// Functions/Basic Container Operations/F_VN_GetAt/F_VN_GetAt_TcVnVector4_UINT

	{attribute 'TcIecLibraryType'}
	{attribute 'external_name' := 'F_VN_GetAt_TcVnVector4_UINT_GUID_DACA282F_CF71_0B71_5078_D95B06B34C79'}
	(* Gets the TcVnVector4_UINT element at the specified index of the container. *)
	FUNCTION F_VN_GetAt_TcVnVector4_UINT : HRESULT
	VAR_INPUT
		ipContainer	:	ITcVnContainer;	(* Container with TcVnVector4_UINT elements *)
		aElement	:	REFERENCE TO TcVnVector4_UINT;	(* Returns the element at the specified index *)
		nIndex	:	ULINT;	(* Index of the requested element *)
		hrPrev	:	HRESULT;	(* HRESULT indicating the result of previous operations (If SUCCEEDED(hrPrev) equals false, no operation is executed.) *)
	END_VAR

END_FUNCTION

// Functions/Basic Container Operations/F_VN_GetAt/F_VN_GetAt_TcVnVector4_USINT

	{attribute 'TcIecLibraryType'}
	{attribute 'external_name' := 'F_VN_GetAt_TcVnVector4_USINT_GUID_B04CDEB5_6B6C_0BE2_4BEB_6EA1CC43E558'}
	(* Gets the TcVnVector4_USINT element at the specified index of the container. *)
	FUNCTION F_VN_GetAt_TcVnVector4_USINT : HRESULT
	VAR_INPUT
		ipContainer	:	ITcVnContainer;	(* Container with TcVnVector4_USINT elements *)
		aElement	:	REFERENCE TO TcVnVector4_USINT;	(* Returns the element at the specified index *)
		nIndex	:	ULINT;	(* Index of the requested element *)
		hrPrev	:	HRESULT;	(* HRESULT indicating the result of previous operations (If SUCCEEDED(hrPrev) equals false, no operation is executed.) *)
	END_VAR

END_FUNCTION

// Functions/Basic Container Operations/F_VN_GetAt/F_VN_GetAt_UDINT

	{attribute 'TcIecLibraryType'}
	{attribute 'external_name' := 'F_VN_GetAt_UDINT_GUID_BF979232_2744_07C5_6489_84B0C61F3275'}
	(* Gets the UDINT element at the specified index of the container. *)
	FUNCTION F_VN_GetAt_UDINT : HRESULT
	VAR_INPUT
		ipContainer	:	ITcVnContainer;	(* Container with UDINT elements *)
		nElement	:	REFERENCE TO UDINT;	(* Returns the element at the specified index *)
		nIndex	:	ULINT;	(* Index of the requested element *)
		hrPrev	:	HRESULT;	(* HRESULT indicating the result of previous operations (If SUCCEEDED(hrPrev) equals false, no operation is executed.) *)
	END_VAR

END_FUNCTION

// Functions/Basic Container Operations/F_VN_GetAt/F_VN_GetAt_UINT

	{attribute 'TcIecLibraryType'}
	{attribute 'external_name' := 'F_VN_GetAt_UINT_GUID_D4F7DF25_3651_0BE4_4285_2E117680DE7D'}
	(* Gets the UINT element at the specified index of the container. *)
	FUNCTION F_VN_GetAt_UINT : HRESULT
	VAR_INPUT
		ipContainer	:	ITcVnContainer;	(* Container with UINT elements *)
		nElement	:	REFERENCE TO UINT;	(* Returns the element at the specified index *)
		nIndex	:	ULINT;	(* Index of the requested element *)
		hrPrev	:	HRESULT;	(* HRESULT indicating the result of previous operations (If SUCCEEDED(hrPrev) equals false, no operation is executed.) *)
	END_VAR

END_FUNCTION

// Functions/Basic Container Operations/F_VN_GetAt/F_VN_GetAt_ULINT

	{attribute 'TcIecLibraryType'}
	{attribute 'external_name' := 'F_VN_GetAt_ULINT_GUID_BCB044E1_AE9F_0A92_654C_54D02EC2BF64'}
	(* Gets the ULINT element at the specified index of the container. *)
	FUNCTION F_VN_GetAt_ULINT : HRESULT
	VAR_INPUT
		ipContainer	:	ITcVnContainer;	(* Container with ULINT elements *)
		nElement	:	REFERENCE TO ULINT;	(* Returns the element at the specified index *)
		nIndex	:	ULINT;	(* Index of the requested element *)
		hrPrev	:	HRESULT;	(* HRESULT indicating the result of previous operations (If SUCCEEDED(hrPrev) equals false, no operation is executed.) *)
	END_VAR

END_FUNCTION

// Functions/Basic Container Operations/F_VN_GetAt/F_VN_GetAt_USINT

	{attribute 'TcIecLibraryType'}
	{attribute 'external_name' := 'F_VN_GetAt_USINT_GUID_3E49D359_324C_0975_751E_A652C8C9EF75'}
	(* Gets the USINT element at the specified index of the container. *)
	FUNCTION F_VN_GetAt_USINT : HRESULT
	VAR_INPUT
		ipContainer	:	ITcVnContainer;	(* Container with USINT elements *)
		nElement	:	REFERENCE TO USINT;	(* Returns the element at the specified index *)
		nIndex	:	ULINT;	(* Index of the requested element *)
		hrPrev	:	HRESULT;	(* HRESULT indicating the result of previous operations (If SUCCEEDED(hrPrev) equals false, no operation is executed.) *)
	END_VAR

END_FUNCTION

// Functions/Basic Container Operations/F_VN_InsertIntoContainer/F_VN_InsertIntoContainer_ITcVnContainer

	{attribute 'TcIecLibraryType'}
	{attribute 'external_name' := 'F_VN_InsertIntoContainer_ITcVnContainer_GUID_A60BDE14_E4D7_0797_570B_140C623D0487'}
	(* Insert an element (or a range of elements) into a container before the specified position. *)
	FUNCTION F_VN_InsertIntoContainer_ITcVnContainer : HRESULT
	VAR_INPUT
		ipElement	:	ITcVnContainer;	(* Single element to insert into ipContainer or container with several elements *)
		ipContainer	:	ITcVnContainer;	(* Container in which to insert the element *)
		nIndex	:	ULINT;	(* Position, before which the element will be inserted *)
		hrPrev	:	HRESULT;	(* HRESULT indicating the result of previous operations (If SUCCEEDED(hrPrev) equals false, no operation is executed.) *)
	END_VAR

END_FUNCTION

// Functions/Basic Container Operations/F_VN_InsertIntoContainer/F_VN_InsertIntoContainer_ITcVnForwardIterator

	{attribute 'TcIecLibraryType'}
	{attribute 'external_name' := 'F_VN_InsertIntoContainer_ITcVnForwardIterator_GUID_FB7539B3_B7C2_0135_5324_E11529024484'}
	(* Insert an element (represented by an iterator) into a container before the specified position. *)
	FUNCTION F_VN_InsertIntoContainer_ITcVnForwardIterator : HRESULT
	VAR_INPUT
		ipElement	:	ITcVnForwardIterator;	(* Single element to insert into ipContainer *)
		ipContainer	:	ITcVnContainer;	(* Container in which to insert the element *)
		nIndex	:	ULINT;	(* Position, before which the element will be inserted *)
		hrPrev	:	HRESULT;	(* HRESULT indicating the result of previous operations (If SUCCEEDED(hrPrev) equals false, no operation is executed.) *)
	END_VAR

END_FUNCTION

// Functions/Basic Container Operations/F_VN_InsertIntoContainer/F_VN_InsertIntoContainer_DINT

	{attribute 'TcIecLibraryType'}
	{attribute 'external_name' := 'F_VN_InsertIntoContainer_DINT_GUID_9477BFDC_23EB_04A7_4507_F78D3CC46D82'}
	(* Insert an element of type DINT into a container before the specified position. *)
	FUNCTION F_VN_InsertIntoContainer_DINT : HRESULT
	VAR_INPUT
		nElement	:	DINT;	(* Single element to insert into ipContainer *)
		ipContainer	:	ITcVnContainer;	(* Container in which to insert the element *)
		nIndex	:	ULINT;	(* Position, before which the element will be inserted *)
		hrPrev	:	HRESULT;	(* HRESULT indicating the result of previous operations (If SUCCEEDED(hrPrev) equals false, no operation is executed.) *)
	END_VAR

END_FUNCTION

// Functions/Basic Container Operations/F_VN_InsertIntoContainer/F_VN_InsertIntoContainer_INT

	{attribute 'TcIecLibraryType'}
	{attribute 'external_name' := 'F_VN_InsertIntoContainer_INT_GUID_6C53FE75_6CDB_00E0_52DC_8EED063716A2'}
	(* Insert an element of type INT into a container before the specified position. *)
	FUNCTION F_VN_InsertIntoContainer_INT : HRESULT
	VAR_INPUT
		nElement	:	INT;	(* Single element to insert into ipContainer *)
		ipContainer	:	ITcVnContainer;	(* Container in which to insert the element *)
		nIndex	:	ULINT;	(* Position, before which the element will be inserted *)
		hrPrev	:	HRESULT;	(* HRESULT indicating the result of previous operations (If SUCCEEDED(hrPrev) equals false, no operation is executed.) *)
	END_VAR

END_FUNCTION

// Functions/Basic Container Operations/F_VN_InsertIntoContainer/F_VN_InsertIntoContainer_ITcVnImage

	{attribute 'TcIecLibraryType'}
	{attribute 'external_name' := 'F_VN_InsertIntoContainer_ITcVnImage_GUID_818AAE11_662C_0FFE_6EFF_8404FD801653'}
	(* Insert an element of type ITcVnImage into a container before the specified position. *)
	FUNCTION F_VN_InsertIntoContainer_ITcVnImage : HRESULT
	VAR_INPUT
		ipElement	:	ITcVnImage;	(* Single element to insert into ipContainer *)
		ipContainer	:	ITcVnContainer;	(* Container in which to insert the element *)
		nIndex	:	ULINT;	(* Position, before which the element will be inserted *)
		hrPrev	:	HRESULT;	(* HRESULT indicating the result of previous operations (If SUCCEEDED(hrPrev) equals false, no operation is executed.) *)
	END_VAR

END_FUNCTION

// Functions/Basic Container Operations/F_VN_InsertIntoContainer/F_VN_InsertIntoContainer_LREAL

	{attribute 'TcIecLibraryType'}
	{attribute 'external_name' := 'F_VN_InsertIntoContainer_LREAL_GUID_096F557A_3F3F_05E3_5F27_949C48CD0B7C'}
	(* Insert an element of type LREAL into a container before the specified position. *)
	FUNCTION F_VN_InsertIntoContainer_LREAL : HRESULT
	VAR_INPUT
		fElement	:	LREAL;	(* Single element to insert into ipContainer *)
		ipContainer	:	ITcVnContainer;	(* Container in which to insert the element *)
		nIndex	:	ULINT;	(* Position, before which the element will be inserted *)
		hrPrev	:	HRESULT;	(* HRESULT indicating the result of previous operations (If SUCCEEDED(hrPrev) equals false, no operation is executed.) *)
	END_VAR

END_FUNCTION

// Functions/Basic Container Operations/F_VN_InsertIntoContainer/F_VN_InsertIntoContainer_REAL

	{attribute 'TcIecLibraryType'}
	{attribute 'external_name' := 'F_VN_InsertIntoContainer_REAL_GUID_45718397_CD8F_043C_4B3C_FAEFC2A76FAA'}
	(* Insert an element of type REAL into a container before the specified position. *)
	FUNCTION F_VN_InsertIntoContainer_REAL : HRESULT
	VAR_INPUT
		fElement	:	REAL;	(* Single element to insert into ipContainer *)
		ipContainer	:	ITcVnContainer;	(* Container in which to insert the element *)
		nIndex	:	ULINT;	(* Position, before which the element will be inserted *)
		hrPrev	:	HRESULT;	(* HRESULT indicating the result of previous operations (If SUCCEEDED(hrPrev) equals false, no operation is executed.) *)
	END_VAR

END_FUNCTION

// Functions/Basic Container Operations/F_VN_InsertIntoContainer/F_VN_InsertIntoContainer_SINT

	{attribute 'TcIecLibraryType'}
	{attribute 'external_name' := 'F_VN_InsertIntoContainer_SINT_GUID_A7FF57E5_5EEA_0357_45DF_3CF7D68E66D8'}
	(* Insert an element of type SINT into a container before the specified position. *)
	FUNCTION F_VN_InsertIntoContainer_SINT : HRESULT
	VAR_INPUT
		nElement	:	SINT;	(* Single element to insert into ipContainer *)
		ipContainer	:	ITcVnContainer;	(* Container in which to insert the element *)
		nIndex	:	ULINT;	(* Position, before which the element will be inserted *)
		hrPrev	:	HRESULT;	(* HRESULT indicating the result of previous operations (If SUCCEEDED(hrPrev) equals false, no operation is executed.) *)
	END_VAR

END_FUNCTION

// Functions/Basic Container Operations/F_VN_InsertIntoContainer/F_VN_InsertIntoContainer_TcVnDMatch

	{attribute 'TcIecLibraryType'}
	{attribute 'external_name' := 'F_VN_InsertIntoContainer_TcVnDMatch_GUID_195FA26A_4C98_0C0C_6341_BCA50298A1E2'}
	(* Insert an element of type TcVnDMatch into a container before the specified position. *)
	FUNCTION F_VN_InsertIntoContainer_TcVnDMatch : HRESULT
	VAR_INPUT
		stElement	:	REFERENCE TO TcVnDMatch;	(* Single element to insert into ipContainer *)
		ipContainer	:	ITcVnContainer;	(* Container in which to insert the element *)
		nIndex	:	ULINT;	(* Position, before which the element will be inserted *)
		hrPrev	:	HRESULT;	(* HRESULT indicating the result of previous operations (If SUCCEEDED(hrPrev) equals false, no operation is executed.) *)
	END_VAR

END_FUNCTION

// Functions/Basic Container Operations/F_VN_InsertIntoContainer/F_VN_InsertIntoContainer_TcVnKeyPoint

	{attribute 'TcIecLibraryType'}
	{attribute 'external_name' := 'F_VN_InsertIntoContainer_TcVnKeyPoint_GUID_CDF375E9_8EF3_01A8_6EAB_4A74123B3E8C'}
	(* Insert an element of type TcVnKeyPoint into a container before the specified position. *)
	FUNCTION F_VN_InsertIntoContainer_TcVnKeyPoint : HRESULT
	VAR_INPUT
		stElement	:	REFERENCE TO TcVnKeyPoint;	(* Single element to insert into ipContainer *)
		ipContainer	:	ITcVnContainer;	(* Container in which to insert the element *)
		nIndex	:	ULINT;	(* Position, before which the element will be inserted *)
		hrPrev	:	HRESULT;	(* HRESULT indicating the result of previous operations (If SUCCEEDED(hrPrev) equals false, no operation is executed.) *)
	END_VAR

END_FUNCTION

// Functions/Basic Container Operations/F_VN_InsertIntoContainer/F_VN_InsertIntoContainer_TcVnPoint2_DINT

	{attribute 'TcIecLibraryType'}
	{attribute 'external_name' := 'F_VN_InsertIntoContainer_TcVnPoint2_DINT_GUID_8E9E8726_B170_0739_7A98_9EC859873B72'}
	(* Insert an element of type TcVnPoint2_DINT into a container before the specified position. *)
	FUNCTION F_VN_InsertIntoContainer_TcVnPoint2_DINT : HRESULT
	VAR_INPUT
		aElement	:	REFERENCE TO TcVnPoint2_DINT;	(* Single element to insert into ipContainer *)
		ipContainer	:	ITcVnContainer;	(* Container in which to insert the element *)
		nIndex	:	ULINT;	(* Position, before which the element will be inserted *)
		hrPrev	:	HRESULT;	(* HRESULT indicating the result of previous operations (If SUCCEEDED(hrPrev) equals false, no operation is executed.) *)
	END_VAR

END_FUNCTION

// Functions/Basic Container Operations/F_VN_InsertIntoContainer/F_VN_InsertIntoContainer_TcVnPoint2_LREAL

	{attribute 'TcIecLibraryType'}
	{attribute 'external_name' := 'F_VN_InsertIntoContainer_TcVnPoint2_LREAL_GUID_74E5ECD1_9927_0D11_6C49_A840E3E3E7C0'}
	(* Insert an element of type TcVnPoint2_LREAL into a container before the specified position. *)
	FUNCTION F_VN_InsertIntoContainer_TcVnPoint2_LREAL : HRESULT
	VAR_INPUT
		aElement	:	REFERENCE TO TcVnPoint2_LREAL;	(* Single element to insert into ipContainer *)
		ipContainer	:	ITcVnContainer;	(* Container in which to insert the element *)
		nIndex	:	ULINT;	(* Position, before which the element will be inserted *)
		hrPrev	:	HRESULT;	(* HRESULT indicating the result of previous operations (If SUCCEEDED(hrPrev) equals false, no operation is executed.) *)
	END_VAR

END_FUNCTION

// Functions/Basic Container Operations/F_VN_InsertIntoContainer/F_VN_InsertIntoContainer_TcVnPoint2_REAL

	{attribute 'TcIecLibraryType'}
	{attribute 'external_name' := 'F_VN_InsertIntoContainer_TcVnPoint2_REAL_GUID_09A8FAC7_C6FC_0592_47AD_1ACE1C999C72'}
	(* Insert an element of type TcVnPoint2_REAL into a container before the specified position. *)
	FUNCTION F_VN_InsertIntoContainer_TcVnPoint2_REAL : HRESULT
	VAR_INPUT
		aElement	:	REFERENCE TO TcVnPoint2_REAL;	(* Single element to insert into ipContainer *)
		ipContainer	:	ITcVnContainer;	(* Container in which to insert the element *)
		nIndex	:	ULINT;	(* Position, before which the element will be inserted *)
		hrPrev	:	HRESULT;	(* HRESULT indicating the result of previous operations (If SUCCEEDED(hrPrev) equals false, no operation is executed.) *)
	END_VAR

END_FUNCTION

// Functions/Basic Container Operations/F_VN_InsertIntoContainer/F_VN_InsertIntoContainer_TcVnPoint3_LREAL

	{attribute 'TcIecLibraryType'}
	{attribute 'external_name' := 'F_VN_InsertIntoContainer_TcVnPoint3_LREAL_GUID_7CA43F0F_BD7B_0D80_4AE2_D06CB9873822'}
	(* Insert an element of type TcVnPoint3_LREAL into a container before the specified position. *)
	FUNCTION F_VN_InsertIntoContainer_TcVnPoint3_LREAL : HRESULT
	VAR_INPUT
		aElement	:	REFERENCE TO TcVnPoint3_LREAL;	(* Single element to insert into ipContainer *)
		ipContainer	:	ITcVnContainer;	(* Container in which to insert the element *)
		nIndex	:	ULINT;	(* Position, before which the element will be inserted *)
		hrPrev	:	HRESULT;	(* HRESULT indicating the result of previous operations (If SUCCEEDED(hrPrev) equals false, no operation is executed.) *)
	END_VAR

END_FUNCTION

// Functions/Basic Container Operations/F_VN_InsertIntoContainer/F_VN_InsertIntoContainer_TcVnPoint3_REAL

	{attribute 'TcIecLibraryType'}
	{attribute 'external_name' := 'F_VN_InsertIntoContainer_TcVnPoint3_REAL_GUID_1DB4729A_8459_030B_6EE4_1D18839BFAC4'}
	(* Insert an element of type TcVnPoint3_REAL into a container before the specified position. *)
	FUNCTION F_VN_InsertIntoContainer_TcVnPoint3_REAL : HRESULT
	VAR_INPUT
		aElement	:	REFERENCE TO TcVnPoint3_REAL;	(* Single element to insert into ipContainer *)
		ipContainer	:	ITcVnContainer;	(* Container in which to insert the element *)
		nIndex	:	ULINT;	(* Position, before which the element will be inserted *)
		hrPrev	:	HRESULT;	(* HRESULT indicating the result of previous operations (If SUCCEEDED(hrPrev) equals false, no operation is executed.) *)
	END_VAR

END_FUNCTION

// Functions/Basic Container Operations/F_VN_InsertIntoContainer/F_VN_InsertIntoContainer_TcVnRectangle_DINT

	{attribute 'TcIecLibraryType'}
	{attribute 'external_name' := 'F_VN_InsertIntoContainer_TcVnRectangle_DINT_GUID_16EB2A49_7769_0D55_564B_599FD1E0CC5C'}
	(* Insert an element of type TcVnRectangle_DINT into a container before the specified position. *)
	FUNCTION F_VN_InsertIntoContainer_TcVnRectangle_DINT : HRESULT
	VAR_INPUT
		stElement	:	REFERENCE TO TcVnRectangle_DINT;	(* Single element to insert into ipContainer *)
		ipContainer	:	ITcVnContainer;	(* Container in which to insert the element *)
		nIndex	:	ULINT;	(* Position, before which the element will be inserted *)
		hrPrev	:	HRESULT;	(* HRESULT indicating the result of previous operations (If SUCCEEDED(hrPrev) equals false, no operation is executed.) *)
	END_VAR

END_FUNCTION

// Functions/Basic Container Operations/F_VN_InsertIntoContainer/F_VN_InsertIntoContainer_TcVnVector2_DINT

	{attribute 'TcIecLibraryType'}
	{attribute 'external_name' := 'F_VN_InsertIntoContainer_TcVnVector2_DINT_GUID_ED047148_33BA_0C1B_5308_9533B5D98312'}
	(* Insert an element of type TcVnVector2_DINT into a container before the specified position. *)
	FUNCTION F_VN_InsertIntoContainer_TcVnVector2_DINT : HRESULT
	VAR_INPUT
		aElement	:	REFERENCE TO TcVnVector2_DINT;	(* Single element to insert into ipContainer *)
		ipContainer	:	ITcVnContainer;	(* Container in which to insert the element *)
		nIndex	:	ULINT;	(* Position, before which the element will be inserted *)
		hrPrev	:	HRESULT;	(* HRESULT indicating the result of previous operations (If SUCCEEDED(hrPrev) equals false, no operation is executed.) *)
	END_VAR

END_FUNCTION

// Functions/Basic Container Operations/F_VN_InsertIntoContainer/F_VN_InsertIntoContainer_TcVnVector2_INT

	{attribute 'TcIecLibraryType'}
	{attribute 'external_name' := 'F_VN_InsertIntoContainer_TcVnVector2_INT_GUID_92266996_E34A_0295_6CE9_2A40BC53C678'}
	(* Insert an element of type TcVnVector2_INT into a container before the specified position. *)
	FUNCTION F_VN_InsertIntoContainer_TcVnVector2_INT : HRESULT
	VAR_INPUT
		aElement	:	REFERENCE TO TcVnVector2_INT;	(* Single element to insert into ipContainer *)
		ipContainer	:	ITcVnContainer;	(* Container in which to insert the element *)
		nIndex	:	ULINT;	(* Position, before which the element will be inserted *)
		hrPrev	:	HRESULT;	(* HRESULT indicating the result of previous operations (If SUCCEEDED(hrPrev) equals false, no operation is executed.) *)
	END_VAR

END_FUNCTION

// Functions/Basic Container Operations/F_VN_InsertIntoContainer/F_VN_InsertIntoContainer_TcVnVector2_REAL

	{attribute 'TcIecLibraryType'}
	{attribute 'external_name' := 'F_VN_InsertIntoContainer_TcVnVector2_REAL_GUID_9C96593E_AD91_0B91_4458_4BAE51CB4067'}
	(* Insert an element of type TcVnVector2_REAL into a container before the specified position. *)
	FUNCTION F_VN_InsertIntoContainer_TcVnVector2_REAL : HRESULT
	VAR_INPUT
		aElement	:	REFERENCE TO TcVnVector2_REAL;	(* Single element to insert into ipContainer *)
		ipContainer	:	ITcVnContainer;	(* Container in which to insert the element *)
		nIndex	:	ULINT;	(* Position, before which the element will be inserted *)
		hrPrev	:	HRESULT;	(* HRESULT indicating the result of previous operations (If SUCCEEDED(hrPrev) equals false, no operation is executed.) *)
	END_VAR

END_FUNCTION

// Functions/Basic Container Operations/F_VN_InsertIntoContainer/F_VN_InsertIntoContainer_TcVnVector2_SINT

	{attribute 'TcIecLibraryType'}
	{attribute 'external_name' := 'F_VN_InsertIntoContainer_TcVnVector2_SINT_GUID_C7C40024_1541_0465_72FC_20CA06C5089E'}
	(* Insert an element of type TcVnVector2_SINT into a container before the specified position. *)
	FUNCTION F_VN_InsertIntoContainer_TcVnVector2_SINT : HRESULT
	VAR_INPUT
		aElement	:	REFERENCE TO TcVnVector2_SINT;	(* Single element to insert into ipContainer *)
		ipContainer	:	ITcVnContainer;	(* Container in which to insert the element *)
		nIndex	:	ULINT;	(* Position, before which the element will be inserted *)
		hrPrev	:	HRESULT;	(* HRESULT indicating the result of previous operations (If SUCCEEDED(hrPrev) equals false, no operation is executed.) *)
	END_VAR

END_FUNCTION

// Functions/Basic Container Operations/F_VN_InsertIntoContainer/F_VN_InsertIntoContainer_TcVnVector2_UINT

	{attribute 'TcIecLibraryType'}
	{attribute 'external_name' := 'F_VN_InsertIntoContainer_TcVnVector2_UINT_GUID_631D15E4_FB39_0F35_58DC_C9FA6CD05CB9'}
	(* Insert an element of type TcVnVector2_UINT into a container before the specified position. *)
	FUNCTION F_VN_InsertIntoContainer_TcVnVector2_UINT : HRESULT
	VAR_INPUT
		aElement	:	REFERENCE TO TcVnVector2_UINT;	(* Single element to insert into ipContainer *)
		ipContainer	:	ITcVnContainer;	(* Container in which to insert the element *)
		nIndex	:	ULINT;	(* Position, before which the element will be inserted *)
		hrPrev	:	HRESULT;	(* HRESULT indicating the result of previous operations (If SUCCEEDED(hrPrev) equals false, no operation is executed.) *)
	END_VAR

END_FUNCTION

// Functions/Basic Container Operations/F_VN_InsertIntoContainer/F_VN_InsertIntoContainer_TcVnVector2_USINT

	{attribute 'TcIecLibraryType'}
	{attribute 'external_name' := 'F_VN_InsertIntoContainer_TcVnVector2_USINT_GUID_E0CF9A89_1354_0085_6748_A626CF644327'}
	(* Insert an element of type TcVnVector2_USINT into a container before the specified position. *)
	FUNCTION F_VN_InsertIntoContainer_TcVnVector2_USINT : HRESULT
	VAR_INPUT
		aElement	:	REFERENCE TO TcVnVector2_USINT;	(* Single element to insert into ipContainer *)
		ipContainer	:	ITcVnContainer;	(* Container in which to insert the element *)
		nIndex	:	ULINT;	(* Position, before which the element will be inserted *)
		hrPrev	:	HRESULT;	(* HRESULT indicating the result of previous operations (If SUCCEEDED(hrPrev) equals false, no operation is executed.) *)
	END_VAR

END_FUNCTION

// Functions/Basic Container Operations/F_VN_InsertIntoContainer/F_VN_InsertIntoContainer_TcVnVector3_INT

	{attribute 'TcIecLibraryType'}
	{attribute 'external_name' := 'F_VN_InsertIntoContainer_TcVnVector3_INT_GUID_2E36832A_2903_0035_56B6_015030D390C5'}
	(* Insert an element of type TcVnVector3_INT into a container before the specified position. *)
	FUNCTION F_VN_InsertIntoContainer_TcVnVector3_INT : HRESULT
	VAR_INPUT
		aElement	:	REFERENCE TO TcVnVector3_INT;	(* Single element to insert into ipContainer *)
		ipContainer	:	ITcVnContainer;	(* Container in which to insert the element *)
		nIndex	:	ULINT;	(* Position, before which the element will be inserted *)
		hrPrev	:	HRESULT;	(* HRESULT indicating the result of previous operations (If SUCCEEDED(hrPrev) equals false, no operation is executed.) *)
	END_VAR

END_FUNCTION

// Functions/Basic Container Operations/F_VN_InsertIntoContainer/F_VN_InsertIntoContainer_TcVnVector3_REAL

	{attribute 'TcIecLibraryType'}
	{attribute 'external_name' := 'F_VN_InsertIntoContainer_TcVnVector3_REAL_GUID_05C67653_0F68_0821_5F2D_B9E49DCABE87'}
	(* Insert an element of type TcVnVector3_REAL into a container before the specified position. *)
	FUNCTION F_VN_InsertIntoContainer_TcVnVector3_REAL : HRESULT
	VAR_INPUT
		aElement	:	REFERENCE TO TcVnVector3_REAL;	(* Single element to insert into ipContainer *)
		ipContainer	:	ITcVnContainer;	(* Container in which to insert the element *)
		nIndex	:	ULINT;	(* Position, before which the element will be inserted *)
		hrPrev	:	HRESULT;	(* HRESULT indicating the result of previous operations (If SUCCEEDED(hrPrev) equals false, no operation is executed.) *)
	END_VAR

END_FUNCTION

// Functions/Basic Container Operations/F_VN_InsertIntoContainer/F_VN_InsertIntoContainer_TcVnVector3_SINT

	{attribute 'TcIecLibraryType'}
	{attribute 'external_name' := 'F_VN_InsertIntoContainer_TcVnVector3_SINT_GUID_176A8E46_759B_0922_6A48_F01C96CBB548'}
	(* Insert an element of type TcVnVector3_SINT into a container before the specified position. *)
	FUNCTION F_VN_InsertIntoContainer_TcVnVector3_SINT : HRESULT
	VAR_INPUT
		aElement	:	REFERENCE TO TcVnVector3_SINT;	(* Single element to insert into ipContainer *)
		ipContainer	:	ITcVnContainer;	(* Container in which to insert the element *)
		nIndex	:	ULINT;	(* Position, before which the element will be inserted *)
		hrPrev	:	HRESULT;	(* HRESULT indicating the result of previous operations (If SUCCEEDED(hrPrev) equals false, no operation is executed.) *)
	END_VAR

END_FUNCTION

// Functions/Basic Container Operations/F_VN_InsertIntoContainer/F_VN_InsertIntoContainer_TcVnVector3_UINT

	{attribute 'TcIecLibraryType'}
	{attribute 'external_name' := 'F_VN_InsertIntoContainer_TcVnVector3_UINT_GUID_2022E372_CCD7_0E1F_5C8E_51F16E5A2DC7'}
	(* Insert an element of type TcVnVector3_UINT into a container before the specified position. *)
	FUNCTION F_VN_InsertIntoContainer_TcVnVector3_UINT : HRESULT
	VAR_INPUT
		aElement	:	REFERENCE TO TcVnVector3_UINT;	(* Single element to insert into ipContainer *)
		ipContainer	:	ITcVnContainer;	(* Container in which to insert the element *)
		nIndex	:	ULINT;	(* Position, before which the element will be inserted *)
		hrPrev	:	HRESULT;	(* HRESULT indicating the result of previous operations (If SUCCEEDED(hrPrev) equals false, no operation is executed.) *)
	END_VAR

END_FUNCTION

// Functions/Basic Container Operations/F_VN_InsertIntoContainer/F_VN_InsertIntoContainer_TcVnVector3_USINT

	{attribute 'TcIecLibraryType'}
	{attribute 'external_name' := 'F_VN_InsertIntoContainer_TcVnVector3_USINT_GUID_49769FC0_A0E4_0479_7E61_3DBD50247039'}
	(* Insert an element of type TcVnVector3_USINT into a container before the specified position. *)
	FUNCTION F_VN_InsertIntoContainer_TcVnVector3_USINT : HRESULT
	VAR_INPUT
		aElement	:	REFERENCE TO TcVnVector3_USINT;	(* Single element to insert into ipContainer *)
		ipContainer	:	ITcVnContainer;	(* Container in which to insert the element *)
		nIndex	:	ULINT;	(* Position, before which the element will be inserted *)
		hrPrev	:	HRESULT;	(* HRESULT indicating the result of previous operations (If SUCCEEDED(hrPrev) equals false, no operation is executed.) *)
	END_VAR

END_FUNCTION

// Functions/Basic Container Operations/F_VN_InsertIntoContainer/F_VN_InsertIntoContainer_TcVnVector4_DINT

	{attribute 'TcIecLibraryType'}
	{attribute 'external_name' := 'F_VN_InsertIntoContainer_TcVnVector4_DINT_GUID_31ED9EF0_3460_0C77_6FD2_D503E33FE09F'}
	(* Insert an element of type TcVnVector4_DINT into a container before the specified position. *)
	FUNCTION F_VN_InsertIntoContainer_TcVnVector4_DINT : HRESULT
	VAR_INPUT
		aElement	:	REFERENCE TO TcVnVector4_DINT;	(* Single element to insert into ipContainer *)
		ipContainer	:	ITcVnContainer;	(* Container in which to insert the element *)
		nIndex	:	ULINT;	(* Position, before which the element will be inserted *)
		hrPrev	:	HRESULT;	(* HRESULT indicating the result of previous operations (If SUCCEEDED(hrPrev) equals false, no operation is executed.) *)
	END_VAR

END_FUNCTION

// Functions/Basic Container Operations/F_VN_InsertIntoContainer/F_VN_InsertIntoContainer_TcVnVector4_INT

	{attribute 'TcIecLibraryType'}
	{attribute 'external_name' := 'F_VN_InsertIntoContainer_TcVnVector4_INT_GUID_ED03A677_D9D2_0DC7_669F_166A5C5BADCD'}
	(* Insert an element of type TcVnVector4_INT into a container before the specified position. *)
	FUNCTION F_VN_InsertIntoContainer_TcVnVector4_INT : HRESULT
	VAR_INPUT
		aElement	:	REFERENCE TO TcVnVector4_INT;	(* Single element to insert into ipContainer *)
		ipContainer	:	ITcVnContainer;	(* Container in which to insert the element *)
		nIndex	:	ULINT;	(* Position, before which the element will be inserted *)
		hrPrev	:	HRESULT;	(* HRESULT indicating the result of previous operations (If SUCCEEDED(hrPrev) equals false, no operation is executed.) *)
	END_VAR

END_FUNCTION

// Functions/Basic Container Operations/F_VN_InsertIntoContainer/F_VN_InsertIntoContainer_TcVnVector4_LREAL

	{attribute 'TcIecLibraryType'}
	{attribute 'external_name' := 'F_VN_InsertIntoContainer_TcVnVector4_LREAL_GUID_7634F334_E86C_0BBF_513A_BF0446A69B05'}
	(* Insert an element of type TcVnVector4_LREAL into a container before the specified position. *)
	FUNCTION F_VN_InsertIntoContainer_TcVnVector4_LREAL : HRESULT
	VAR_INPUT
		aElement	:	REFERENCE TO TcVnVector4_LREAL;	(* Single element to insert into ipContainer *)
		ipContainer	:	ITcVnContainer;	(* Container in which to insert the element *)
		nIndex	:	ULINT;	(* Position, before which the element will be inserted *)
		hrPrev	:	HRESULT;	(* HRESULT indicating the result of previous operations (If SUCCEEDED(hrPrev) equals false, no operation is executed.) *)
	END_VAR

END_FUNCTION

// Functions/Basic Container Operations/F_VN_InsertIntoContainer/F_VN_InsertIntoContainer_TcVnVector4_SINT

	{attribute 'TcIecLibraryType'}
	{attribute 'external_name' := 'F_VN_InsertIntoContainer_TcVnVector4_SINT_GUID_6DFD1BE3_02B8_0EB9_72A9_DE2F3C302CFF'}
	(* Insert an element of type TcVnVector4_SINT into a container before the specified position. *)
	FUNCTION F_VN_InsertIntoContainer_TcVnVector4_SINT : HRESULT
	VAR_INPUT
		aElement	:	REFERENCE TO TcVnVector4_SINT;	(* Single element to insert into ipContainer *)
		ipContainer	:	ITcVnContainer;	(* Container in which to insert the element *)
		nIndex	:	ULINT;	(* Position, before which the element will be inserted *)
		hrPrev	:	HRESULT;	(* HRESULT indicating the result of previous operations (If SUCCEEDED(hrPrev) equals false, no operation is executed.) *)
	END_VAR

END_FUNCTION

// Functions/Basic Container Operations/F_VN_InsertIntoContainer/F_VN_InsertIntoContainer_TcVnVector4_UINT

	{attribute 'TcIecLibraryType'}
	{attribute 'external_name' := 'F_VN_InsertIntoContainer_TcVnVector4_UINT_GUID_DACF4562_17BE_0AA0_71C5_1DFFBC06FC0F'}
	(* Insert an element of type TcVnVector4_UINT into a container before the specified position. *)
	FUNCTION F_VN_InsertIntoContainer_TcVnVector4_UINT : HRESULT
	VAR_INPUT
		aElement	:	REFERENCE TO TcVnVector4_UINT;	(* Single element to insert into ipContainer *)
		ipContainer	:	ITcVnContainer;	(* Container in which to insert the element *)
		nIndex	:	ULINT;	(* Position, before which the element will be inserted *)
		hrPrev	:	HRESULT;	(* HRESULT indicating the result of previous operations (If SUCCEEDED(hrPrev) equals false, no operation is executed.) *)
	END_VAR

END_FUNCTION

// Functions/Basic Container Operations/F_VN_InsertIntoContainer/F_VN_InsertIntoContainer_TcVnVector4_USINT

	{attribute 'TcIecLibraryType'}
	{attribute 'external_name' := 'F_VN_InsertIntoContainer_TcVnVector4_USINT_GUID_057AB20F_A675_0771_7557_D744E69E14B5'}
	(* Insert an element of type TcVnVector4_USINT into a container before the specified position. *)
	FUNCTION F_VN_InsertIntoContainer_TcVnVector4_USINT : HRESULT
	VAR_INPUT
		aElement	:	REFERENCE TO TcVnVector4_USINT;	(* Single element to insert into ipContainer *)
		ipContainer	:	ITcVnContainer;	(* Container in which to insert the element *)
		nIndex	:	ULINT;	(* Position, before which the element will be inserted *)
		hrPrev	:	HRESULT;	(* HRESULT indicating the result of previous operations (If SUCCEEDED(hrPrev) equals false, no operation is executed.) *)
	END_VAR

END_FUNCTION

// Functions/Basic Container Operations/F_VN_InsertIntoContainer/F_VN_InsertIntoContainer_UDINT

	{attribute 'TcIecLibraryType'}
	{attribute 'external_name' := 'F_VN_InsertIntoContainer_UDINT_GUID_CD06AF6D_CC22_002D_6F10_E76DA43683F9'}
	(* Insert an element of type UDINT into a container before the specified position. *)
	FUNCTION F_VN_InsertIntoContainer_UDINT : HRESULT
	VAR_INPUT
		nElement	:	UDINT;	(* Single element to insert into ipContainer *)
		ipContainer	:	ITcVnContainer;	(* Container in which to insert the element *)
		nIndex	:	ULINT;	(* Position, before which the element will be inserted *)
		hrPrev	:	HRESULT;	(* HRESULT indicating the result of previous operations (If SUCCEEDED(hrPrev) equals false, no operation is executed.) *)
	END_VAR

END_FUNCTION

// Functions/Basic Container Operations/F_VN_InsertIntoContainer/F_VN_InsertIntoContainer_UINT

	{attribute 'TcIecLibraryType'}
	{attribute 'external_name' := 'F_VN_InsertIntoContainer_UINT_GUID_E32B6997_7644_0B75_6DBE_2D469527BD7A'}
	(* Insert an element of type UINT into a container before the specified position. *)
	FUNCTION F_VN_InsertIntoContainer_UINT : HRESULT
	VAR_INPUT
		nElement	:	UINT;	(* Single element to insert into ipContainer *)
		ipContainer	:	ITcVnContainer;	(* Container in which to insert the element *)
		nIndex	:	ULINT;	(* Position, before which the element will be inserted *)
		hrPrev	:	HRESULT;	(* HRESULT indicating the result of previous operations (If SUCCEEDED(hrPrev) equals false, no operation is executed.) *)
	END_VAR

END_FUNCTION

// Functions/Basic Container Operations/F_VN_InsertIntoContainer/F_VN_InsertIntoContainer_ULINT

	{attribute 'TcIecLibraryType'}
	{attribute 'external_name' := 'F_VN_InsertIntoContainer_ULINT_GUID_767FC602_60A6_018C_6D0F_B08EB0072409'}
	(* Insert an element of type ULINT into a container before the specified position. *)
	FUNCTION F_VN_InsertIntoContainer_ULINT : HRESULT
	VAR_INPUT
		nElement	:	ULINT;	(* Single element to insert into ipContainer *)
		ipContainer	:	ITcVnContainer;	(* Container in which to insert the element *)
		nIndex	:	ULINT;	(* Position, before which the element will be inserted *)
		hrPrev	:	HRESULT;	(* HRESULT indicating the result of previous operations (If SUCCEEDED(hrPrev) equals false, no operation is executed.) *)
	END_VAR

END_FUNCTION

// Functions/Basic Container Operations/F_VN_InsertIntoContainer/F_VN_InsertIntoContainer_USINT

	{attribute 'TcIecLibraryType'}
	{attribute 'external_name' := 'F_VN_InsertIntoContainer_USINT_GUID_203DB5BB_AF96_0E43_4CC3_88C1C1B80281'}
	(* Insert an element of type USINT into a container before the specified position. *)
	FUNCTION F_VN_InsertIntoContainer_USINT : HRESULT
	VAR_INPUT
		nElement	:	USINT;	(* Single element to insert into ipContainer *)
		ipContainer	:	ITcVnContainer;	(* Container in which to insert the element *)
		nIndex	:	ULINT;	(* Position, before which the element will be inserted *)
		hrPrev	:	HRESULT;	(* HRESULT indicating the result of previous operations (If SUCCEEDED(hrPrev) equals false, no operation is executed.) *)
	END_VAR

END_FUNCTION

// Functions/Basic Container Operations/F_VN_SetAt/F_VN_SetAt_ITcVnContainer

	{attribute 'TcIecLibraryType'}
	{attribute 'external_name' := 'F_VN_SetAt_ITcVnContainer_GUID_3CB5DB29_E3A8_0807_5C29_ACD6807211B9'}
	(* Sets the element at the specified index of the container. (Alternatively use interface method .SetAt.) *)
	FUNCTION F_VN_SetAt_ITcVnContainer : HRESULT
	VAR_INPUT
		ipElement	:	ITcVnContainer;	(* Element to set at the specified container position *)
		ipContainer	:	ITcVnContainer;	(* Container with ITcVnContainer elements, in which the element at position nIndex is replaced by ipElement *)
		nIndex	:	ULINT;	(* Index *)
		hrPrev	:	HRESULT;	(* HRESULT indicating the result of previous operations (If SUCCEEDED(hrPrev) equals false, no operation is executed.) *)
	END_VAR

END_FUNCTION

// Functions/Basic Container Operations/F_VN_SetAt/F_VN_SetAt_DINT

	{attribute 'TcIecLibraryType'}
	{attribute 'external_name' := 'F_VN_SetAt_DINT_GUID_AD568E0B_CD2F_08DA_63B7_4E5BC66002AE'}
	(* Sets the element at the specified index of the container. *)
	FUNCTION F_VN_SetAt_DINT : HRESULT
	VAR_INPUT
		nElement	:	DINT;	(* Element to set at the specified container position *)
		ipContainer	:	ITcVnContainer;	(* Container with DINT elements, in which the element at position nIndex is replaced by nElement *)
		nIndex	:	ULINT;	(* Index *)
		hrPrev	:	HRESULT;	(* HRESULT indicating the result of previous operations (If SUCCEEDED(hrPrev) equals false, no operation is executed.) *)
	END_VAR

END_FUNCTION

// Functions/Basic Container Operations/F_VN_SetAt/F_VN_SetAt_INT

	{attribute 'TcIecLibraryType'}
	{attribute 'external_name' := 'F_VN_SetAt_INT_GUID_38804B15_FD1F_0705_4E0D_3D63332CF396'}
	(* Sets the element at the specified index of the container. *)
	FUNCTION F_VN_SetAt_INT : HRESULT
	VAR_INPUT
		nElement	:	INT;	(* Element to set at the specified container position *)
		ipContainer	:	ITcVnContainer;	(* Container with INT elements, in which the element at position nIndex is replaced by nElement *)
		nIndex	:	ULINT;	(* Index *)
		hrPrev	:	HRESULT;	(* HRESULT indicating the result of previous operations (If SUCCEEDED(hrPrev) equals false, no operation is executed.) *)
	END_VAR

END_FUNCTION

// Functions/Basic Container Operations/F_VN_SetAt/F_VN_SetAt_ITcVnImage

	{attribute 'TcIecLibraryType'}
	{attribute 'external_name' := 'F_VN_SetAt_ITcVnImage_GUID_039F3365_758F_0FF4_4E4B_978FAAACAB8B'}
	(* Sets the element at the specified index of the container. *)
	FUNCTION F_VN_SetAt_ITcVnImage : HRESULT
	VAR_INPUT
		ipElement	:	ITcVnImage;	(* Element to set at the specified container position *)
		ipContainer	:	ITcVnContainer;	(* Container with ITcVnImage elements, in which the element at position nIndex is replaced by ipElement *)
		nIndex	:	ULINT;	(* Index *)
		hrPrev	:	HRESULT;	(* HRESULT indicating the result of previous operations (If SUCCEEDED(hrPrev) equals false, no operation is executed.) *)
	END_VAR

END_FUNCTION

// Functions/Basic Container Operations/F_VN_SetAt/F_VN_SetAt_LREAL

	{attribute 'TcIecLibraryType'}
	{attribute 'external_name' := 'F_VN_SetAt_LREAL_GUID_39E11F5F_6A3F_0C38_6059_AD55062C95CE'}
	(* Sets the element at the specified index of the container. *)
	FUNCTION F_VN_SetAt_LREAL : HRESULT
	VAR_INPUT
		fElement	:	LREAL;	(* Element to set at the specified container position *)
		ipContainer	:	ITcVnContainer;	(* Container with LREAL elements, in which the element at position nIndex is replaced by fElement *)
		nIndex	:	ULINT;	(* Index *)
		hrPrev	:	HRESULT;	(* HRESULT indicating the result of previous operations (If SUCCEEDED(hrPrev) equals false, no operation is executed.) *)
	END_VAR

END_FUNCTION

// Functions/Basic Container Operations/F_VN_SetAt/F_VN_SetAt_REAL

	{attribute 'TcIecLibraryType'}
	{attribute 'external_name' := 'F_VN_SetAt_REAL_GUID_F6F7C1AA_76E6_0056_7520_73D2A2845852'}
	(* Sets the element at the specified index of the container. *)
	FUNCTION F_VN_SetAt_REAL : HRESULT
	VAR_INPUT
		fElement	:	REAL;	(* Element to set at the specified container position *)
		ipContainer	:	ITcVnContainer;	(* Container with REAL elements, in which the element at position nIndex is replaced by fElement *)
		nIndex	:	ULINT;	(* Index *)
		hrPrev	:	HRESULT;	(* HRESULT indicating the result of previous operations (If SUCCEEDED(hrPrev) equals false, no operation is executed.) *)
	END_VAR

END_FUNCTION

// Functions/Basic Container Operations/F_VN_SetAt/F_VN_SetAt_SINT

	{attribute 'TcIecLibraryType'}
	{attribute 'external_name' := 'F_VN_SetAt_SINT_GUID_282B3FB8_E285_01FA_5DC3_ED6CAEA8ECE8'}
	(* Sets the element at the specified index of the container. *)
	FUNCTION F_VN_SetAt_SINT : HRESULT
	VAR_INPUT
		nElement	:	SINT;	(* Element to set at the specified container position *)
		ipContainer	:	ITcVnContainer;	(* Container with SINT elements, in which the element at position nIndex is replaced by nElement *)
		nIndex	:	ULINT;	(* Index *)
		hrPrev	:	HRESULT;	(* HRESULT indicating the result of previous operations (If SUCCEEDED(hrPrev) equals false, no operation is executed.) *)
	END_VAR

END_FUNCTION

// Functions/Basic Container Operations/F_VN_SetAt/F_VN_SetAt_TcVnDMatch

	{attribute 'TcIecLibraryType'}
	{attribute 'external_name' := 'F_VN_SetAt_TcVnDMatch_GUID_A5B43D48_6061_06EC_4520_B87470DCA5CF'}
	(* Sets the element at the specified index of the container. *)
	FUNCTION F_VN_SetAt_TcVnDMatch : HRESULT
	VAR_INPUT
		stElement	:	REFERENCE TO TcVnDMatch;	(* Element to set at the specified container position *)
		ipContainer	:	ITcVnContainer;	(* Container with TcVnDMatch elements, in which the element at position nIndex is replaced by stElement *)
		nIndex	:	ULINT;	(* Index *)
		hrPrev	:	HRESULT;	(* HRESULT indicating the result of previous operations (If SUCCEEDED(hrPrev) equals false, no operation is executed.) *)
	END_VAR

END_FUNCTION

// Functions/Basic Container Operations/F_VN_SetAt/F_VN_SetAt_TcVnKeyPoint

	{attribute 'TcIecLibraryType'}
	{attribute 'external_name' := 'F_VN_SetAt_TcVnKeyPoint_GUID_DD200FE0_9133_0AA4_5E82_EACEC4FD0853'}
	(* Sets the element at the specified index of the container. *)
	FUNCTION F_VN_SetAt_TcVnKeyPoint : HRESULT
	VAR_INPUT
		stElement	:	REFERENCE TO TcVnKeyPoint;	(* Element to set at the specified container position *)
		ipContainer	:	ITcVnContainer;	(* Container with TcVnKeyPoint elements, in which the element at position nIndex is replaced by stElement *)
		nIndex	:	ULINT;	(* Index *)
		hrPrev	:	HRESULT;	(* HRESULT indicating the result of previous operations (If SUCCEEDED(hrPrev) equals false, no operation is executed.) *)
	END_VAR

END_FUNCTION

// Functions/Basic Container Operations/F_VN_SetAt/F_VN_SetAt_TcVnPoint2_DINT

	{attribute 'TcIecLibraryType'}
	{attribute 'external_name' := 'F_VN_SetAt_TcVnPoint2_DINT_GUID_B06E87E8_4C32_0670_603F_B3B5939761DB'}
	(* Sets the element at the specified index of the container. *)
	FUNCTION F_VN_SetAt_TcVnPoint2_DINT : HRESULT
	VAR_INPUT
		aElement	:	REFERENCE TO TcVnPoint2_DINT;	(* Element to set at the specified container position *)
		ipContainer	:	ITcVnContainer;	(* Container with TcVnPoint2_DINT elements, in which the element at position nIndex is replaced by aElement *)
		nIndex	:	ULINT;	(* Index *)
		hrPrev	:	HRESULT;	(* HRESULT indicating the result of previous operations (If SUCCEEDED(hrPrev) equals false, no operation is executed.) *)
	END_VAR

END_FUNCTION

// Functions/Basic Container Operations/F_VN_SetAt/F_VN_SetAt_TcVnPoint2_LREAL

	{attribute 'TcIecLibraryType'}
	{attribute 'external_name' := 'F_VN_SetAt_TcVnPoint2_LREAL_GUID_BB5772DD_0ADE_0511_7845_0FA397D78F14'}
	(* Sets the element at the specified index of the container. *)
	FUNCTION F_VN_SetAt_TcVnPoint2_LREAL : HRESULT
	VAR_INPUT
		aElement	:	REFERENCE TO TcVnPoint2_LREAL;	(* Element to set at the specified container position *)
		ipContainer	:	ITcVnContainer;	(* Container with TcVnPoint2_LREAL elements, in which the element at position nIndex is replaced by aElement *)
		nIndex	:	ULINT;	(* Index *)
		hrPrev	:	HRESULT;	(* HRESULT indicating the result of previous operations (If SUCCEEDED(hrPrev) equals false, no operation is executed.) *)
	END_VAR

END_FUNCTION

// Functions/Basic Container Operations/F_VN_SetAt/F_VN_SetAt_TcVnPoint2_REAL

	{attribute 'TcIecLibraryType'}
	{attribute 'external_name' := 'F_VN_SetAt_TcVnPoint2_REAL_GUID_EB5EEA43_B839_0954_439D_6DBABC0A42E4'}
	(* Sets the element at the specified index of the container. *)
	FUNCTION F_VN_SetAt_TcVnPoint2_REAL : HRESULT
	VAR_INPUT
		aElement	:	REFERENCE TO TcVnPoint2_REAL;	(* Element to set at the specified container position *)
		ipContainer	:	ITcVnContainer;	(* Container with TcVnPoint2_REAL elements, in which the element at position nIndex is replaced by aElement *)
		nIndex	:	ULINT;	(* Index *)
		hrPrev	:	HRESULT;	(* HRESULT indicating the result of previous operations (If SUCCEEDED(hrPrev) equals false, no operation is executed.) *)
	END_VAR

END_FUNCTION

// Functions/Basic Container Operations/F_VN_SetAt/F_VN_SetAt_TcVnPoint3_LREAL

	{attribute 'TcIecLibraryType'}
	{attribute 'external_name' := 'F_VN_SetAt_TcVnPoint3_LREAL_GUID_7264CF52_FDAE_044E_4B08_5C8668A93908'}
	(* Sets the element at the specified index of the container. *)
	FUNCTION F_VN_SetAt_TcVnPoint3_LREAL : HRESULT
	VAR_INPUT
		aElement	:	REFERENCE TO TcVnPoint3_LREAL;	(* Element to set at the specified container position *)
		ipContainer	:	ITcVnContainer;	(* Container with TcVnPoint3_LREAL elements, in which the element at position nIndex is replaced by aElement *)
		nIndex	:	ULINT;	(* Index *)
		hrPrev	:	HRESULT;	(* HRESULT indicating the result of previous operations (If SUCCEEDED(hrPrev) equals false, no operation is executed.) *)
	END_VAR

END_FUNCTION

// Functions/Basic Container Operations/F_VN_SetAt/F_VN_SetAt_TcVnPoint3_REAL

	{attribute 'TcIecLibraryType'}
	{attribute 'external_name' := 'F_VN_SetAt_TcVnPoint3_REAL_GUID_4171A4CD_80E5_0B4D_7100_9339127026C8'}
	(* Sets the element at the specified index of the container. *)
	FUNCTION F_VN_SetAt_TcVnPoint3_REAL : HRESULT
	VAR_INPUT
		aElement	:	REFERENCE TO TcVnPoint3_REAL;	(* Element to set at the specified container position *)
		ipContainer	:	ITcVnContainer;	(* Container with TcVnPoint3_REAL elements, in which the element at position nIndex is replaced by aElement *)
		nIndex	:	ULINT;	(* Index *)
		hrPrev	:	HRESULT;	(* HRESULT indicating the result of previous operations (If SUCCEEDED(hrPrev) equals false, no operation is executed.) *)
	END_VAR

END_FUNCTION

// Functions/Basic Container Operations/F_VN_SetAt/F_VN_SetAt_TcVnRectangle_DINT

	{attribute 'TcIecLibraryType'}
	{attribute 'external_name' := 'F_VN_SetAt_TcVnRectangle_DINT_GUID_CD501511_0376_0F0C_5163_BE0C3FBF2C29'}
	(* Sets the element at the specified index of the container. *)
	FUNCTION F_VN_SetAt_TcVnRectangle_DINT : HRESULT
	VAR_INPUT
		stElement	:	REFERENCE TO TcVnRectangle_DINT;	(* Element to set at the specified container position *)
		ipContainer	:	ITcVnContainer;	(* Container with TcVnRectangle_DINT elements, in which the element at position nIndex is replaced by stElement *)
		nIndex	:	ULINT;	(* Index *)
		hrPrev	:	HRESULT;	(* HRESULT indicating the result of previous operations (If SUCCEEDED(hrPrev) equals false, no operation is executed.) *)
	END_VAR

END_FUNCTION

// Functions/Basic Container Operations/F_VN_SetAt/F_VN_SetAt_TcVnVector2_DINT

	{attribute 'TcIecLibraryType'}
	{attribute 'external_name' := 'F_VN_SetAt_TcVnVector2_DINT_GUID_A6FEF05D_4B73_0528_6EB9_24AE5AF5221E'}
	(* Sets the element at the specified index of the container. *)
	FUNCTION F_VN_SetAt_TcVnVector2_DINT : HRESULT
	VAR_INPUT
		aElement	:	REFERENCE TO TcVnVector2_DINT;	(* Element to set at the specified container position *)
		ipContainer	:	ITcVnContainer;	(* Container with TcVnVector2_DINT elements, in which the element at position nIndex is replaced by aElement *)
		nIndex	:	ULINT;	(* Index *)
		hrPrev	:	HRESULT;	(* HRESULT indicating the result of previous operations (If SUCCEEDED(hrPrev) equals false, no operation is executed.) *)
	END_VAR

END_FUNCTION

// Functions/Basic Container Operations/F_VN_SetAt/F_VN_SetAt_TcVnVector2_INT

	{attribute 'TcIecLibraryType'}
	{attribute 'external_name' := 'F_VN_SetAt_TcVnVector2_INT_GUID_62A89D97_FFB0_0713_73CF_8AE6D7FA7A9E'}
	(* Sets the element at the specified index of the container. *)
	FUNCTION F_VN_SetAt_TcVnVector2_INT : HRESULT
	VAR_INPUT
		aElement	:	REFERENCE TO TcVnVector2_INT;	(* Element to set at the specified container position *)
		ipContainer	:	ITcVnContainer;	(* Container with TcVnVector2_INT elements, in which the element at position nIndex is replaced by aElement *)
		nIndex	:	ULINT;	(* Index *)
		hrPrev	:	HRESULT;	(* HRESULT indicating the result of previous operations (If SUCCEEDED(hrPrev) equals false, no operation is executed.) *)
	END_VAR

END_FUNCTION

// Functions/Basic Container Operations/F_VN_SetAt/F_VN_SetAt_TcVnVector2_REAL

	{attribute 'TcIecLibraryType'}
	{attribute 'external_name' := 'F_VN_SetAt_TcVnVector2_REAL_GUID_748C4431_4054_039E_6A93_FB230551FD79'}
	(* Sets the element at the specified index of the container. *)
	FUNCTION F_VN_SetAt_TcVnVector2_REAL : HRESULT
	VAR_INPUT
		aElement	:	REFERENCE TO TcVnVector2_REAL;	(* Element to set at the specified container position *)
		ipContainer	:	ITcVnContainer;	(* Container with TcVnVector2_REAL elements, in which the element at position nIndex is replaced by aElement *)
		nIndex	:	ULINT;	(* Index *)
		hrPrev	:	HRESULT;	(* HRESULT indicating the result of previous operations (If SUCCEEDED(hrPrev) equals false, no operation is executed.) *)
	END_VAR

END_FUNCTION

// Functions/Basic Container Operations/F_VN_SetAt/F_VN_SetAt_TcVnVector2_SINT

	{attribute 'TcIecLibraryType'}
	{attribute 'external_name' := 'F_VN_SetAt_TcVnVector2_SINT_GUID_B91EF4FE_F266_0BC9_4674_322B83DD367D'}
	(* Sets the element at the specified index of the container. *)
	FUNCTION F_VN_SetAt_TcVnVector2_SINT : HRESULT
	VAR_INPUT
		aElement	:	REFERENCE TO TcVnVector2_SINT;	(* Element to set at the specified container position *)
		ipContainer	:	ITcVnContainer;	(* Container with TcVnVector2_SINT elements, in which the element at position nIndex is replaced by aElement *)
		nIndex	:	ULINT;	(* Index *)
		hrPrev	:	HRESULT;	(* HRESULT indicating the result of previous operations (If SUCCEEDED(hrPrev) equals false, no operation is executed.) *)
	END_VAR

END_FUNCTION

// Functions/Basic Container Operations/F_VN_SetAt/F_VN_SetAt_TcVnVector2_UINT

	{attribute 'TcIecLibraryType'}
	{attribute 'external_name' := 'F_VN_SetAt_TcVnVector2_UINT_GUID_D902C69B_5D69_0647_6366_E19D48240ADA'}
	(* Sets the element at the specified index of the container. *)
	FUNCTION F_VN_SetAt_TcVnVector2_UINT : HRESULT
	VAR_INPUT
		aElement	:	REFERENCE TO TcVnVector2_UINT;	(* Element to set at the specified container position *)
		ipContainer	:	ITcVnContainer;	(* Container with TcVnVector2_UINT elements, in which the element at position nIndex is replaced by aElement *)
		nIndex	:	ULINT;	(* Index *)
		hrPrev	:	HRESULT;	(* HRESULT indicating the result of previous operations (If SUCCEEDED(hrPrev) equals false, no operation is executed.) *)
	END_VAR

END_FUNCTION

// Functions/Basic Container Operations/F_VN_SetAt/F_VN_SetAt_TcVnVector2_USINT

	{attribute 'TcIecLibraryType'}
	{attribute 'external_name' := 'F_VN_SetAt_TcVnVector2_USINT_GUID_899B786E_0D5E_05FA_78AB_D00D84BD0067'}
	(* Sets the element at the specified index of the container. *)
	FUNCTION F_VN_SetAt_TcVnVector2_USINT : HRESULT
	VAR_INPUT
		aElement	:	REFERENCE TO TcVnVector2_USINT;	(* Element to set at the specified container position *)
		ipContainer	:	ITcVnContainer;	(* Container with TcVnVector2_USINT elements, in which the element at position nIndex is replaced by aElement *)
		nIndex	:	ULINT;	(* Index *)
		hrPrev	:	HRESULT;	(* HRESULT indicating the result of previous operations (If SUCCEEDED(hrPrev) equals false, no operation is executed.) *)
	END_VAR

END_FUNCTION

// Functions/Basic Container Operations/F_VN_SetAt/F_VN_SetAt_TcVnVector3_INT

	{attribute 'TcIecLibraryType'}
	{attribute 'external_name' := 'F_VN_SetAt_TcVnVector3_INT_GUID_4B7BA833_0A48_02CE_4C4D_CA84535647C5'}
	(* Sets the element at the specified index of the container. *)
	FUNCTION F_VN_SetAt_TcVnVector3_INT : HRESULT
	VAR_INPUT
		aElement	:	REFERENCE TO TcVnVector3_INT;	(* Element to set at the specified container position *)
		ipContainer	:	ITcVnContainer;	(* Container with TcVnVector3_INT elements, in which the element at position nIndex is replaced by aElement *)
		nIndex	:	ULINT;	(* Index *)
		hrPrev	:	HRESULT;	(* HRESULT indicating the result of previous operations (If SUCCEEDED(hrPrev) equals false, no operation is executed.) *)
	END_VAR

END_FUNCTION

// Functions/Basic Container Operations/F_VN_SetAt/F_VN_SetAt_TcVnVector3_REAL

	{attribute 'TcIecLibraryType'}
	{attribute 'external_name' := 'F_VN_SetAt_TcVnVector3_REAL_GUID_6F83B025_52D6_079F_6A92_2E3CCDB23C02'}
	(* Sets the element at the specified index of the container. *)
	FUNCTION F_VN_SetAt_TcVnVector3_REAL : HRESULT
	VAR_INPUT
		aElement	:	REFERENCE TO TcVnVector3_REAL;	(* Element to set at the specified container position *)
		ipContainer	:	ITcVnContainer;	(* Container with TcVnVector3_REAL elements, in which the element at position nIndex is replaced by aElement *)
		nIndex	:	ULINT;	(* Index *)
		hrPrev	:	HRESULT;	(* HRESULT indicating the result of previous operations (If SUCCEEDED(hrPrev) equals false, no operation is executed.) *)
	END_VAR

END_FUNCTION

// Functions/Basic Container Operations/F_VN_SetAt/F_VN_SetAt_TcVnVector3_SINT

	{attribute 'TcIecLibraryType'}
	{attribute 'external_name' := 'F_VN_SetAt_TcVnVector3_SINT_GUID_7A380888_B654_09B2_5EED_ECB2FE5A6BB9'}
	(* Sets the element at the specified index of the container. *)
	FUNCTION F_VN_SetAt_TcVnVector3_SINT : HRESULT
	VAR_INPUT
		aElement	:	REFERENCE TO TcVnVector3_SINT;	(* Element to set at the specified container position *)
		ipContainer	:	ITcVnContainer;	(* Container with TcVnVector3_SINT elements, in which the element at position nIndex is replaced by aElement *)
		nIndex	:	ULINT;	(* Index *)
		hrPrev	:	HRESULT;	(* HRESULT indicating the result of previous operations (If SUCCEEDED(hrPrev) equals false, no operation is executed.) *)
	END_VAR

END_FUNCTION

// Functions/Basic Container Operations/F_VN_SetAt/F_VN_SetAt_TcVnVector3_UINT

	{attribute 'TcIecLibraryType'}
	{attribute 'external_name' := 'F_VN_SetAt_TcVnVector3_UINT_GUID_488854F4_215E_0443_7EC6_EDD5A2686F29'}
	(* Sets the element at the specified index of the container. *)
	FUNCTION F_VN_SetAt_TcVnVector3_UINT : HRESULT
	VAR_INPUT
		aElement	:	REFERENCE TO TcVnVector3_UINT;	(* Element to set at the specified container position *)
		ipContainer	:	ITcVnContainer;	(* Container with TcVnVector3_UINT elements, in which the element at position nIndex is replaced by aElement *)
		nIndex	:	ULINT;	(* Index *)
		hrPrev	:	HRESULT;	(* HRESULT indicating the result of previous operations (If SUCCEEDED(hrPrev) equals false, no operation is executed.) *)
	END_VAR

END_FUNCTION

// Functions/Basic Container Operations/F_VN_SetAt/F_VN_SetAt_TcVnVector3_USINT

	{attribute 'TcIecLibraryType'}
	{attribute 'external_name' := 'F_VN_SetAt_TcVnVector3_USINT_GUID_32644D7E_48A5_0093_7871_3A8C252AA3D1'}
	(* Sets the element at the specified index of the container. *)
	FUNCTION F_VN_SetAt_TcVnVector3_USINT : HRESULT
	VAR_INPUT
		aElement	:	REFERENCE TO TcVnVector3_USINT;	(* Element to set at the specified container position *)
		ipContainer	:	ITcVnContainer;	(* Container with TcVnVector3_USINT elements, in which the element at position nIndex is replaced by aElement *)
		nIndex	:	ULINT;	(* Index *)
		hrPrev	:	HRESULT;	(* HRESULT indicating the result of previous operations (If SUCCEEDED(hrPrev) equals false, no operation is executed.) *)
	END_VAR

END_FUNCTION

// Functions/Basic Container Operations/F_VN_SetAt/F_VN_SetAt_TcVnVector4_DINT

	{attribute 'TcIecLibraryType'}
	{attribute 'external_name' := 'F_VN_SetAt_TcVnVector4_DINT_GUID_7CFB044D_CF29_0355_75D7_4B90455C3C33'}
	(* Sets the element at the specified index of the container. *)
	FUNCTION F_VN_SetAt_TcVnVector4_DINT : HRESULT
	VAR_INPUT
		aElement	:	REFERENCE TO TcVnVector4_DINT;	(* Element to set at the specified container position *)
		ipContainer	:	ITcVnContainer;	(* Container with TcVnVector4_DINT elements, in which the element at position nIndex is replaced by aElement *)
		nIndex	:	ULINT;	(* Index *)
		hrPrev	:	HRESULT;	(* HRESULT indicating the result of previous operations (If SUCCEEDED(hrPrev) equals false, no operation is executed.) *)
	END_VAR

END_FUNCTION

// Functions/Basic Container Operations/F_VN_SetAt/F_VN_SetAt_TcVnVector4_INT

	{attribute 'TcIecLibraryType'}
	{attribute 'external_name' := 'F_VN_SetAt_TcVnVector4_INT_GUID_B47A9F71_A1C0_0B76_7617_854A00A2708A'}
	(* Sets the element at the specified index of the container. *)
	FUNCTION F_VN_SetAt_TcVnVector4_INT : HRESULT
	VAR_INPUT
		aElement	:	REFERENCE TO TcVnVector4_INT;	(* Element to set at the specified container position *)
		ipContainer	:	ITcVnContainer;	(* Container with TcVnVector4_INT elements, in which the element at position nIndex is replaced by aElement *)
		nIndex	:	ULINT;	(* Index *)
		hrPrev	:	HRESULT;	(* HRESULT indicating the result of previous operations (If SUCCEEDED(hrPrev) equals false, no operation is executed.) *)
	END_VAR

END_FUNCTION

// Functions/Basic Container Operations/F_VN_SetAt/F_VN_SetAt_TcVnVector4_LREAL

	{attribute 'TcIecLibraryType'}
	{attribute 'external_name' := 'F_VN_SetAt_TcVnVector4_LREAL_GUID_4B7D1F48_28E8_0A90_7DCC_DB2E7C77127F'}
	(* Sets the element at the specified index of the container. *)
	FUNCTION F_VN_SetAt_TcVnVector4_LREAL : HRESULT
	VAR_INPUT
		aElement	:	REFERENCE TO TcVnVector4_LREAL;	(* Element to set at the specified container position *)
		ipContainer	:	ITcVnContainer;	(* Container with TcVnVector4_LREAL elements, in which the element at position nIndex is replaced by aElement *)
		nIndex	:	ULINT;	(* Index *)
		hrPrev	:	HRESULT;	(* HRESULT indicating the result of previous operations (If SUCCEEDED(hrPrev) equals false, no operation is executed.) *)
	END_VAR

END_FUNCTION

// Functions/Basic Container Operations/F_VN_SetAt/F_VN_SetAt_TcVnVector4_SINT

	{attribute 'TcIecLibraryType'}
	{attribute 'external_name' := 'F_VN_SetAt_TcVnVector4_SINT_GUID_62D8C98D_C1B4_0D51_471A_82A25FBEB769'}
	(* Sets the element at the specified index of the container. *)
	FUNCTION F_VN_SetAt_TcVnVector4_SINT : HRESULT
	VAR_INPUT
		aElement	:	REFERENCE TO TcVnVector4_SINT;	(* Element to set at the specified container position *)
		ipContainer	:	ITcVnContainer;	(* Container with TcVnVector4_SINT elements, in which the element at position nIndex is replaced by aElement *)
		nIndex	:	ULINT;	(* Index *)
		hrPrev	:	HRESULT;	(* HRESULT indicating the result of previous operations (If SUCCEEDED(hrPrev) equals false, no operation is executed.) *)
	END_VAR

END_FUNCTION

// Functions/Basic Container Operations/F_VN_SetAt/F_VN_SetAt_TcVnVector4_UINT

	{attribute 'TcIecLibraryType'}
	{attribute 'external_name' := 'F_VN_SetAt_TcVnVector4_UINT_GUID_64806559_95F2_06F8_5D17_50A269732263'}
	(* Sets the element at the specified index of the container. *)
	FUNCTION F_VN_SetAt_TcVnVector4_UINT : HRESULT
	VAR_INPUT
		aElement	:	REFERENCE TO TcVnVector4_UINT;	(* Element to set at the specified container position *)
		ipContainer	:	ITcVnContainer;	(* Container with TcVnVector4_UINT elements, in which the element at position nIndex is replaced by aElement *)
		nIndex	:	ULINT;	(* Index *)
		hrPrev	:	HRESULT;	(* HRESULT indicating the result of previous operations (If SUCCEEDED(hrPrev) equals false, no operation is executed.) *)
	END_VAR

END_FUNCTION

// Functions/Basic Container Operations/F_VN_SetAt/F_VN_SetAt_TcVnVector4_USINT

	{attribute 'TcIecLibraryType'}
	{attribute 'external_name' := 'F_VN_SetAt_TcVnVector4_USINT_GUID_74379A52_7BAB_04AD_6407_AEF21A12DE18'}
	(* Sets the element at the specified index of the container. *)
	FUNCTION F_VN_SetAt_TcVnVector4_USINT : HRESULT
	VAR_INPUT
		aElement	:	REFERENCE TO TcVnVector4_USINT;	(* Element to set at the specified container position *)
		ipContainer	:	ITcVnContainer;	(* Container with TcVnVector4_USINT elements, in which the element at position nIndex is replaced by aElement *)
		nIndex	:	ULINT;	(* Index *)
		hrPrev	:	HRESULT;	(* HRESULT indicating the result of previous operations (If SUCCEEDED(hrPrev) equals false, no operation is executed.) *)
	END_VAR

END_FUNCTION

// Functions/Basic Container Operations/F_VN_SetAt/F_VN_SetAt_UDINT

	{attribute 'TcIecLibraryType'}
	{attribute 'external_name' := 'F_VN_SetAt_UDINT_GUID_3B671B11_C3E8_0138_7382_0DA88D45D321'}
	(* Sets the element at the specified index of the container. *)
	FUNCTION F_VN_SetAt_UDINT : HRESULT
	VAR_INPUT
		nElement	:	UDINT;	(* Element to set at the specified container position *)
		ipContainer	:	ITcVnContainer;	(* Container with UDINT elements, in which the element at position nIndex is replaced by nElement *)
		nIndex	:	ULINT;	(* Index *)
		hrPrev	:	HRESULT;	(* HRESULT indicating the result of previous operations (If SUCCEEDED(hrPrev) equals false, no operation is executed.) *)
	END_VAR

END_FUNCTION

// Functions/Basic Container Operations/F_VN_SetAt/F_VN_SetAt_UINT

	{attribute 'TcIecLibraryType'}
	{attribute 'external_name' := 'F_VN_SetAt_UINT_GUID_6FC150F1_84AD_0ECF_505A_772F3BFFB85A'}
	(* Sets the element at the specified index of the container. *)
	FUNCTION F_VN_SetAt_UINT : HRESULT
	VAR_INPUT
		nElement	:	UINT;	(* Element to set at the specified container position *)
		ipContainer	:	ITcVnContainer;	(* Container with UINT elements, in which the element at position nIndex is replaced by nElement *)
		nIndex	:	ULINT;	(* Index *)
		hrPrev	:	HRESULT;	(* HRESULT indicating the result of previous operations (If SUCCEEDED(hrPrev) equals false, no operation is executed.) *)
	END_VAR

END_FUNCTION

// Functions/Basic Container Operations/F_VN_SetAt/F_VN_SetAt_ULINT

	{attribute 'TcIecLibraryType'}
	{attribute 'external_name' := 'F_VN_SetAt_ULINT_GUID_04744F62_D332_024E_4E21_1295A3B7BFAF'}
	(* Sets the element at the specified index of the container. *)
	FUNCTION F_VN_SetAt_ULINT : HRESULT
	VAR_INPUT
		nElement	:	ULINT;	(* Element to set at the specified container position *)
		ipContainer	:	ITcVnContainer;	(* Container with ULINT elements, in which the element at position nIndex is replaced by nElement *)
		nIndex	:	ULINT;	(* Index *)
		hrPrev	:	HRESULT;	(* HRESULT indicating the result of previous operations (If SUCCEEDED(hrPrev) equals false, no operation is executed.) *)
	END_VAR

END_FUNCTION

// Functions/Basic Container Operations/F_VN_SetAt/F_VN_SetAt_USINT

	{attribute 'TcIecLibraryType'}
	{attribute 'external_name' := 'F_VN_SetAt_USINT_GUID_899B094C_1051_0518_52EA_9F7207A72ED2'}
	(* Sets the element at the specified index of the container. *)
	FUNCTION F_VN_SetAt_USINT : HRESULT
	VAR_INPUT
		nElement	:	USINT;	(* Element to set at the specified container position *)
		ipContainer	:	ITcVnContainer;	(* Container with USINT elements, in which the element at position nIndex is replaced by nElement *)
		nIndex	:	ULINT;	(* Index *)
		hrPrev	:	HRESULT;	(* HRESULT indicating the result of previous operations (If SUCCEEDED(hrPrev) equals false, no operation is executed.) *)
	END_VAR

END_FUNCTION

// Functions/Geometric and Coordinate Transformations/Calibration/F_VN_CalibrateCamera

	{attribute 'TcIecLibraryType'}
	{attribute 'external_name' := 'F_VN_CalibrateCamera_GUID_134D0641_6B58_0E5F_5E31_6AF62A8328B8'}
	(* Compute the camera parameters (intrinsic + extrinsic) by evaluating an image containing a calibration pattern (circles). *)
	FUNCTION F_VN_CalibrateCamera : HRESULT
	VAR_INPUT
		ipSrcImage	:	ITcVnImage;	(* Source image containing a calibration pattern (1 channel, USINT elements) *)
		ipReferencePoints	:	ITcVnContainer;	(* Reference calibration pattern point positions (ContainerType_Vector_TcVnPoint3_REAL) *)
		aCameraMatrix	:	REFERENCE TO TcVnMatrix3x3_LREAL;	(* Returns the camera matrix *)
		aDistortionCoefficients	:	REFERENCE TO TcVnArray8_LREAL;	(* Returns the lens distortion coefficients [k1, k2, p1, p2, k3, k4, k5, k6] *)
		aRotationMatrix	:	REFERENCE TO TcVnMatrix3x3_LREAL;	(* Returns the rotation matrix *)
		aTranslationVector	:	REFERENCE TO TcVnVector3_LREAL;	(* Returns the translation vector *)
		fReprojError	:	REFERENCE TO LREAL;	(* Returns the reprojection error *)
		stBlobDetectionParams	:	REFERENCE TO TcVnParamsBlobDetection;	(* Parameters for the internally used F_VN_DetectBlobs function *)
		stCalibrationOptions	:	REFERENCE TO TcVnCameraCalibrationOptions;	(* Calibration options *)
		hrPrev	:	HRESULT;	(* HRESULT indicating the result of previous operations (If SUCCEEDED(hrPrev) equals false, no operation is executed.) *)
	END_VAR

END_FUNCTION

// Functions/Geometric and Coordinate Transformations/Calibration/F_VN_CalibrateCameraExp

	{attribute 'TcIecLibraryType'}
	{attribute 'external_name' := 'F_VN_CalibrateCameraExp_GUID_E598C6A8_9CC3_0105_45E9_4E69F516739E'}
	(* Compute the camera parameters (intrinsic + extrinsic) by evaluating images containing a calibration pattern (circles). The extrinsic parameters are computed for the first image in the array. (expert function) *)
	FUNCTION F_VN_CalibrateCameraExp : HRESULT
	VAR_INPUT
		pSrcImages	:	PVOID;	(* Pointer to an array of source images, each containing the same calibration pattern (1 channel, USINT elements) *)
		nSrcArraySize	:	UINT;	(* pSrcImages array size *)
		ipReferencePoints	:	ITcVnContainer;	(* Reference calibration pattern point positions (ContainerType_Vector_TcVnPoint3_REAL) *)
		aCameraMatrix	:	REFERENCE TO TcVnMatrix3x3_LREAL;	(* Returns the camera matrix *)
		aDistortionCoefficients	:	REFERENCE TO TcVnArray8_LREAL;	(* Returns the lens distortion coefficients [k1, k2, p1, p2, k3, k4, k5, k6] *)
		aRotationMatrix	:	REFERENCE TO TcVnMatrix3x3_LREAL;	(* Returns the rotation matrix *)
		aTranslationVector	:	REFERENCE TO TcVnVector3_LREAL;	(* Returns the translation vector *)
		fReprojError	:	REFERENCE TO LREAL;	(* Returns the reprojection error *)
		stBlobDetectionParams	:	REFERENCE TO TcVnParamsBlobDetection;	(* Parameters for the internally used F_VN_DetectBlobs function *)
		stCalibrationOptions	:	REFERENCE TO TcVnCameraCalibrationOptions;	(* Calibration options *)
		hrPrev	:	HRESULT;	(* HRESULT indicating the result of previous operations (If SUCCEEDED(hrPrev) equals false, no operation is executed.) *)
	END_VAR

END_FUNCTION

// Functions/Geometric and Coordinate Transformations/Calibration/F_VN_CalibrateCameraExp2

	{attribute 'TcIecLibraryType'}
	{attribute 'external_name' := 'F_VN_CalibrateCameraExp2_GUID_717D6D44_E183_03E3_60AF_ABF44C1D7471'}
	(* Compute the camera parameters (intrinsic + extrinsic) by evaluating images containing a calibration pattern (circles). The extrinsic parameters are computed for the first image in the array. (expert function) *)
	FUNCTION F_VN_CalibrateCameraExp2 : HRESULT
	VAR_INPUT
		pSrcImages	:	PVOID;	(* Pointer to an array of source images, each containing the same calibration pattern (1 channel, USINT elements) *)
		nSrcArraySize	:	UINT;	(* pSrcImages array size *)
		ipReferencePoints	:	ITcVnContainer;	(* Reference calibration pattern point positions (ContainerType_Vector_TcVnPoint3_REAL) *)
		aCameraMatrix	:	REFERENCE TO TcVnMatrix3x3_LREAL;	(* Returns the camera matrix *)
		aDistortionCoefficients	:	REFERENCE TO TcVnArray8_LREAL;	(* Returns the lens distortion coefficients [k1, k2, p1, p2, k3, k4, k5, k6] *)
		aRotationMatrix	:	REFERENCE TO TcVnMatrix3x3_LREAL;	(* Returns the rotation matrix *)
		aTranslationVector	:	REFERENCE TO TcVnVector3_LREAL;	(* Returns the translation vector *)
		fReprojError	:	REFERENCE TO LREAL;	(* Returns the reprojection error *)
		stBlobDetectionParams	:	REFERENCE TO TcVnParamsBlobDetection;	(* Parameters for the internally used F_VN_DetectBlobs function *)
		stCalibrationOptions	:	REFERENCE TO TcVnCameraCalibrationOptions;	(* Calibration options *)
		bSubpixelAccuracy	:	BOOL;	(* If true, the pattern points are detected with subpixel accuracy *)
		eEdgeDirection	:	ETcVnEdgeDirection;	(* Specification of the edge direction to search for (from center to outside ellipse) *)
		fMinStrength	:	REAL;	(* Specification of the minimum strength (intensity difference) of the edge to search for *)
		nMaxThickness	:	UDINT;	(* Specification of the maximum thickness of the edge to search for, which means fMinStrength must be reached within nMaxThickness pixels *)
		nSubpixelsIterations	:	UDINT;	(* Specifies the number of subpixels (for INTERPOLATION, 10 - 20 usually is sufficient) or maximum number of iterations for optimizing the parameters (for APPROX_ERF and APPROX_GAUSSIAN, 50 - 100 usually is sufficient) *)
		nSearchLines	:	UDINT;	(* Specifies the amount of search lines, which are equally distributed in all directions (must be >= 8 and a multiple of 4) *)
		fApproxPrecision	:	REAL;	(* Specifies the approximation precision for APPROX_ERF and APPROX_GAUSSIAN (0.001 usually is sufficient, unused for INTERPOLATION) *)
		eAlgorithm	:	ETcVnEdgeDetectionAlgorithm;	(* Selection of the edge detection algorithm *)
		hrPrev	:	HRESULT;	(* HRESULT indicating the result of previous operations (If SUCCEEDED(hrPrev) equals false, no operation is executed.) *)
	END_VAR

END_FUNCTION

// Functions/Geometric and Coordinate Transformations/Calibration/F_VN_CalibrateCameraExp3

	{attribute 'TcIecLibraryType'}
	{attribute 'external_name' := 'F_VN_CalibrateCameraExp3_GUID_210F9815_03C2_0D92_4CD1_07AAD29B87DB'}
	(* Compute the camera parameters (intrinsic + extrinsic) by evaluating images containing a calibration pattern (circles). The extrinsic parameters are computed for the first image in the array. (expert function) *)
	FUNCTION F_VN_CalibrateCameraExp3 : HRESULT
	VAR_INPUT
		pSrcImages	:	PVOID;	(* Pointer to an array of source images, each containing the same calibration pattern (1 channel, USINT elements) *)
		nSrcArraySize	:	UINT;	(* pSrcImages array size *)
		ipReferencePoints	:	ITcVnContainer;	(* Reference calibration pattern point positions (ContainerType_Vector_TcVnPoint3_REAL) *)
		aCameraMatrix	:	REFERENCE TO TcVnMatrix3x3_LREAL;	(* Returns the camera matrix *)
		aDistortionCoefficients	:	REFERENCE TO TcVnArray8_LREAL;	(* Returns the lens distortion coefficients [k1, k2, p1, p2, k3, k4, k5, k6] *)
		aRotationMatrix	:	REFERENCE TO TcVnMatrix3x3_LREAL;	(* Returns the rotation matrix *)
		aTranslationVector	:	REFERENCE TO TcVnVector3_LREAL;	(* Returns the translation vector *)
		fReprojError	:	REFERENCE TO LREAL;	(* Returns the reprojection error *)
		stBlobDetectionParams	:	REFERENCE TO TcVnParamsBlobDetection;	(* Parameters for the internally used F_VN_DetectBlobs function *)
		stCalibrationOptions	:	REFERENCE TO TcVnCameraCalibrationOptions;	(* Calibration options *)
		bSubpixelAccuracy	:	BOOL;	(* If true, the pattern points are detected with subpixel accuracy *)
		eEdgeDirection	:	ETcVnEdgeDirection;	(* Specification of the edge direction to search for (from center to outside ellipse) *)
		fMinStrength	:	REAL;	(* Specification of the minimum strength (intensity difference) of the edge to search for *)
		nMaxThickness	:	UDINT;	(* Specification of the maximum thickness of the edge to search for, which means fMinStrength must be reached within nMaxThickness pixels *)
		nSubpixelsIterations	:	UDINT;	(* Specifies the number of subpixels (for INTERPOLATION, 10 - 20 usually is sufficient) or maximum number of iterations for optimizing the parameters (for APPROX_ERF and APPROX_GAUSSIAN, 50 - 100 usually is sufficient) *)
		nSearchLines	:	UDINT;	(* Specifies the amount of search lines, which are equally distributed in all directions (must be >= 8 and a multiple of 4) *)
		fApproxPrecision	:	REAL;	(* Specifies the approximation precision for APPROX_ERF and APPROX_GAUSSIAN (0.001 usually is sufficient, unused for INTERPOLATION) *)
		eAlgorithm	:	ETcVnEdgeDetectionAlgorithm;	(* Selection of the edge detection algorithm *)
		eWorldSystem	:	ETcVnWorldCoordinateSystem;	(* World coordinate system orientation *)
		hrPrev	:	HRESULT;	(* HRESULT indicating the result of previous operations (If SUCCEEDED(hrPrev) equals false, no operation is executed.) *)
	END_VAR

END_FUNCTION

// Functions/Geometric and Coordinate Transformations/Calibration/F_VN_CalibrateCameraManually

	{attribute 'TcIecLibraryType'}
	{attribute 'external_name' := 'F_VN_CalibrateCameraManually_GUID_A55F542E_2B4C_0AF8_5989_1940328F1C22'}
	(* Compute the camera parameters (intrinsic + extrinsic). The extrinsic parameters are computed for the first inner container. *)
	FUNCTION F_VN_CalibrateCameraManually : HRESULT
	VAR_INPUT
		ipImagePoints	:	ITcVnContainer;	(* Provided image points of multiple images (ContainerType_Vector_Vector_TcVnPoint2_REAL, each inner container with at least 6 points). The container and point order must match ipReferencePoints. *)
		nImageWidth	:	UDINT;	(* Image width *)
		nImageHeight	:	UDINT;	(* Image height *)
		ipReferencePoints	:	ITcVnContainer;	(* Reference world points (ContainerType_Vector_Vector_TcVnPoint3_REAL). The number of inner containers and their amount of points must match ipImagePoints. *)
		aCameraMatrix	:	REFERENCE TO TcVnMatrix3x3_LREAL;	(* Returns the camera matrix *)
		aDistortionCoefficients	:	REFERENCE TO TcVnArray8_LREAL;	(* Returns the lens distortion coefficients [k1, k2, p1, p2, k3, k4, k5, k6] *)
		aRotationMatrix	:	REFERENCE TO TcVnMatrix3x3_LREAL;	(* Returns the rotation matrix (for the first inner container) *)
		aTranslationVector	:	REFERENCE TO TcVnVector3_LREAL;	(* Returns the translation vector (for the first inner container) *)
		fReprojError	:	REFERENCE TO LREAL;	(* Returns the reprojection error *)
		stCalibrationOptions	:	REFERENCE TO TcVnCameraCalibrationOptions;	(* Calibration options *)
		hrPrev	:	HRESULT;	(* HRESULT indicating the result of previous operations (If SUCCEEDED(hrPrev) equals false, no operation is executed.) *)
	END_VAR

END_FUNCTION

// Functions/Geometric and Coordinate Transformations/Calibration/F_VN_CalibrateCameraManuallyExp

	{attribute 'TcIecLibraryType'}
	{attribute 'external_name' := 'F_VN_CalibrateCameraManuallyExp_GUID_26313ECD_99ED_03D2_55A2_6F00B2FF78F0'}
	(* Compute the camera parameters (intrinsic + extrinsic). The extrinsic parameters are computed for the first inner container. (expert function) *)
	FUNCTION F_VN_CalibrateCameraManuallyExp : HRESULT
	VAR_INPUT
		ipImagePoints	:	ITcVnContainer;	(* Provided image points of multiple images (ContainerType_Vector_Vector_TcVnPoint2_REAL, each inner container with at least 6 points). The container and point order must match ipReferencePoints. *)
		nImageWidth	:	UDINT;	(* Image width *)
		nImageHeight	:	UDINT;	(* Image height *)
		ipReferencePoints	:	ITcVnContainer;	(* Reference world points (ContainerType_Vector_Vector_TcVnPoint3_REAL). The number of inner containers and their amount of points must match ipImagePoints. *)
		aCameraMatrix	:	REFERENCE TO TcVnMatrix3x3_LREAL;	(* Returns the camera matrix *)
		aDistortionCoefficients	:	REFERENCE TO TcVnArray8_LREAL;	(* Returns the lens distortion coefficients [k1, k2, p1, p2, k3, k4, k5, k6] *)
		aRotationMatrix	:	REFERENCE TO TcVnMatrix3x3_LREAL;	(* Returns the rotation matrix (for the first inner container) *)
		aTranslationVector	:	REFERENCE TO TcVnVector3_LREAL;	(* Returns the translation vector (for the first inner container) *)
		fReprojError	:	REFERENCE TO LREAL;	(* Returns the reprojection error *)
		stCalibrationOptions	:	REFERENCE TO TcVnCameraCalibrationOptions;	(* Calibration options *)
		eWorldSystem	:	ETcVnWorldCoordinateSystem;	(* World coordinate system orientation *)
		hrPrev	:	HRESULT;	(* HRESULT indicating the result of previous operations (If SUCCEEDED(hrPrev) equals false, no operation is executed.) *)
	END_VAR

END_FUNCTION

// Functions/Geometric and Coordinate Transformations/Calibration/F_VN_CalibrateCameraPlanar

	{attribute 'TcIecLibraryType'}
	{attribute 'external_name' := 'F_VN_CalibrateCameraPlanar_GUID_257158C4_BCB2_04D1_7159_524970C8B55A'}
	(* Calibrate camera using a planar calibration pattern comprised of four circles marking the corners of a rectangle. *)
	FUNCTION F_VN_CalibrateCameraPlanar : HRESULT
	VAR_INPUT
		ipSrcImage	:	ITcVnImage;	(* Binary source image (background zero, markers non-zero) *)
		aMarkerPositions	:	REFERENCE TO TcVnArray4_Point2_REAL;	(* Marker positions within their plane using world units (right-handed coordinate system) *)
		aTransformationMatrix	:	REFERENCE TO TcVnMatrix3x3_LREAL;	(* Returns a 3-by-3 matrix for the transformation from image coordinates into the reference coordinate system *)
		hrPrev	:	HRESULT;	(* HRESULT indicating the result of previous operations (If SUCCEEDED(hrPrev) equals false, no operation is executed.) *)
	END_VAR

END_FUNCTION

// Functions/Geometric and Coordinate Transformations/Calibration/F_VN_CalibrateCameraPlanarExp

	{attribute 'TcIecLibraryType'}
	{attribute 'external_name' := 'F_VN_CalibrateCameraPlanarExp_GUID_85168C06_73E8_09D6_648F_BFAE58F27DE2'}
	(* Calibrate camera using a planar calibration pattern comprised of four circles marking the corners of a rectangle. (expert function) *)
	FUNCTION F_VN_CalibrateCameraPlanarExp : HRESULT
	VAR_INPUT
		ipSrcImage	:	ITcVnImage;	(* Binary source image (background zero, markers non-zero) *)
		aMarkerPositions	:	REFERENCE TO TcVnArray4_Point2_REAL;	(* Marker positions within their plane using world units (right-handed coordinate system) *)
		aTransformationMatrix	:	REFERENCE TO TcVnMatrix3x3_LREAL;	(* Returns a 3-by-3 matrix for the transformation from image coordinates into the reference coordinate system *)
		aMarkerImagePositions	:	REFERENCE TO TcVnArray4_Point2_REAL;	(* Returns the marker positions in image coordinates (left-handed coordinate system) *)
		nMinMarkerArea	:	UDINT;	(* Minimum area for the detection of markers (Smaller markers are ignored.) *)
		nMaxMarkerArea	:	UDINT;	(* Maximum area for the detection of markers (Larger markers are ignored.) *)
		fMaxMarkerEccentricity	:	LREAL;	(* Maximum eccenticity for the detection of markers (The eccentricity measures deviations from a round shape (eccentricity = 0: round object; eccentricity = 1.0:  linear object).) *)
		hrPrev	:	HRESULT;	(* HRESULT indicating the result of previous operations (If SUCCEEDED(hrPrev) equals false, no operation is executed.) *)
	END_VAR

END_FUNCTION

// Functions/Geometric and Coordinate Transformations/Calibration/F_VN_CalibrateLinescanCamera

	{attribute 'TcIecLibraryType'}
	{attribute 'external_name' := 'F_VN_CalibrateLinescanCamera_GUID_78F7EB50_74BC_0971_7AFB_D12F932FB047'}
	(* Compute the camera parameters (intrinsic + extrinsic) by evaluating images containing a line calibration pattern, consisting of alternating vertical and diagonal lines, each diagonal line having the same constant slope: |\|\|...\|. To be compatible to 2d calibration results, the y-position of the image line is set to half sensor width, so that it would be the center line of a virtual 2d sensor with equal width and height. The extrinsic parameters are computed for the first image in the array. *)
	FUNCTION F_VN_CalibrateLinescanCamera : HRESULT
	VAR_INPUT
		pSrcImages	:	PVOID;	(* Pointer to an array of 1 or more source images (1 channel). If the images have more than 1 row, each row must contain an image of the same pattern position. *)
		nSrcArraySize	:	UINT;	(* pSrcImages array size *)
		ipPatternLineOrigins	:	ITcVnContainer;	(* X position of the pattern line origins (ContainerType_Vector_REAL, usually same origin for vertical and following diagonal line) *)
		fSlopeRad	:	LREAL;	(* Slope of the diagonal line in rad (> 0, < PI/2), relative to the vertical line (i.e., 0 would be a vertical line, PI/2 a horizontal line) *)
		aCameraMatrix	:	REFERENCE TO TcVnMatrix3x3_LREAL;	(* Returns the camera matrix *)
		aDistortionCoefficients	:	REFERENCE TO TcVnArray8_LREAL;	(* Returns the lens distortion coefficients [k1, k2, p1, p2, k3, k4, k5, k6] *)
		aRotationMatrix	:	REFERENCE TO TcVnMatrix3x3_LREAL;	(* Returns the rotation matrix *)
		aTranslationVector	:	REFERENCE TO TcVnVector3_LREAL;	(* Returns the translation vector *)
		fReprojError	:	REFERENCE TO LREAL;	(* Returns the reprojection error *)
		stCalibrationOptions	:	REFERENCE TO TcVnCameraCalibrationOptions;	(* Calibration options (recommended to set bFixAspectRatio, bFixPrincipalPoint, bZeroTangentDist) *)
		eEdgeDirection	:	ETcVnEdgeDirection;	(* Specification of the edge direction to search for *)
		hrPrev	:	HRESULT;	(* HRESULT indicating the result of previous operations (If SUCCEEDED(hrPrev) equals false, no operation is executed.) *)
	END_VAR

END_FUNCTION

// Functions/Geometric and Coordinate Transformations/Calibration/F_VN_CalibrateLinescanCameraExp

	{attribute 'TcIecLibraryType'}
	{attribute 'external_name' := 'F_VN_CalibrateLinescanCameraExp_GUID_559B40D7_42F6_0CA2_5248_382F82F67F26'}
	(* Compute the camera parameters (intrinsic + extrinsic) by evaluating images containing a line calibration pattern, consisting of alternating vertical and diagonal lines, each diagonal line having the same constant slope: |\|\|...\|. To be compatible to 2d calibration results, the y-position of the image line is set to half sensor width, so that it would be the center line of a virtual 2d sensor with equal width and height. The extrinsic parameters are computed for the first image in the array. (expert function) *)
	FUNCTION F_VN_CalibrateLinescanCameraExp : HRESULT
	VAR_INPUT
		pSrcImages	:	PVOID;	(* Pointer to an array of 1 or more source images (1 channel). If the images have more than 1 row, each row must contain an image of the same pattern position. *)
		nSrcArraySize	:	UINT;	(* pSrcImages array size *)
		ipPatternLineOrigins	:	ITcVnContainer;	(* X position of the pattern line origins (ContainerType_Vector_REAL, usually same origin for vertical and following diagonal line) *)
		fSlopeRad	:	LREAL;	(* Slope of the diagonal line in rad (> 0, < PI/2), relative to the vertical line (i.e., 0 would be a vertical line, PI/2 a horizontal line) *)
		aCameraMatrix	:	REFERENCE TO TcVnMatrix3x3_LREAL;	(* Returns the camera matrix *)
		aDistortionCoefficients	:	REFERENCE TO TcVnArray8_LREAL;	(* Returns the lens distortion coefficients [k1, k2, p1, p2, k3, k4, k5, k6] *)
		aRotationMatrix	:	REFERENCE TO TcVnMatrix3x3_LREAL;	(* Returns the rotation matrix *)
		aTranslationVector	:	REFERENCE TO TcVnVector3_LREAL;	(* Returns the translation vector *)
		fReprojError	:	REFERENCE TO LREAL;	(* Returns the reprojection error *)
		stCalibrationOptions	:	REFERENCE TO TcVnCameraCalibrationOptions;	(* Calibration options (recommended to set bFixAspectRatio, bFixPrincipalPoint, bZeroTangentDist) *)
		eEdgeDirection	:	ETcVnEdgeDirection;	(* Specification of the edge direction to search for *)
		fMinStrength	:	REAL;	(* Specification of the minimum strength (intensity difference) of the edge to search for *)
		nMaxSearchLines	:	UDINT;	(* Maximum number of search lines (equally distributed over the image height, at most 1 searchline per image row) *)
		nMaxThickness	:	UDINT;	(* Specification of the maximum thickness of the edge to search for, which means fMinStrength must be reached within nMaxThickness pixels *)
		nSubpixelsIterations	:	UDINT;	(* Specifies the number of subpixels (for INTERPOLATION, 10 - 20 usually is sufficient) or maximum number of iterations for optimizing the parameters (for APPROX_ERF and APPROX_GAUSSIAN, 50 - 100 usually is sufficient) *)
		fApproxPrecision	:	REAL;	(* Specifies the approximation precision for APPROX_ERF and APPROX_GAUSSIAN (0.001 usually is sufficient, unused for INTERPOLATION) *)
		eAlgorithm	:	ETcVnEdgeDetectionAlgorithm;	(* Selection of the edge detection algorithm *)
		hrPrev	:	HRESULT;	(* HRESULT indicating the result of previous operations (If SUCCEEDED(hrPrev) equals false, no operation is executed.) *)
	END_VAR

END_FUNCTION

// Functions/Geometric and Coordinate Transformations/Calibration/F_VN_CompensateLensDistortion

	{attribute 'TcIecLibraryType'}
	{attribute 'external_name' := 'F_VN_CompensateLensDistortion_GUID_B066A958_2635_07C8_4D61_92F5FBA7F883'}
	(* Transforms an image to compensate the lens distortion. *)
	FUNCTION F_VN_CompensateLensDistortion : HRESULT
	VAR_INPUT
		ipSrcImage	:	ITcVnImage;	(* Source image *)
		ipDestImage	:	REFERENCE TO ITcVnImage;	(* Destination image (An appropriate destination image will be created if required.) *)
		aCameraMatrix	:	REFERENCE TO TcVnMatrix3x3_LREAL;	(* Camera matrix containing the intrinsic parameters *)
		aDistortionCoefficients	:	REFERENCE TO TcVnArray4_LREAL;	(* Lens distortion coefficients [k1, k2, p1, p2] *)
		hrPrev	:	HRESULT;	(* HRESULT indicating the result of previous operations (If SUCCEEDED(hrPrev) equals false, no operation is executed.) *)
	END_VAR

END_FUNCTION

// Functions/Geometric and Coordinate Transformations/Calibration/F_VN_CompensateLensDistortionExp1

	{attribute 'TcIecLibraryType'}
	{attribute 'external_name' := 'F_VN_CompensateLensDistortionExp1_GUID_2A1BCF5F_7A16_0BD3_4AF5_8530BAFFC403'}
	(* Transforms an image to compensate the lens distortion. (expert function) *)
	FUNCTION F_VN_CompensateLensDistortionExp1 : HRESULT
	VAR_INPUT
		ipSrcImage	:	ITcVnImage;	(* Source image *)
		ipDestImage	:	REFERENCE TO ITcVnImage;	(* Destination image (An appropriate destination image will be created if required.) *)
		aCameraMatrix	:	REFERENCE TO TcVnMatrix3x3_LREAL;	(* Camera matrix containing the intrinsic parameters *)
		aDistortionCoefficients	:	REFERENCE TO TcVnArray8_LREAL;	(* Lens distortion coefficients [k1, k2, p1, p2, k3, k4, k5, k6] *)
		hrPrev	:	HRESULT;	(* HRESULT indicating the result of previous operations (If SUCCEEDED(hrPrev) equals false, no operation is executed.) *)
	END_VAR

END_FUNCTION

// Functions/Geometric and Coordinate Transformations/Calibration/F_VN_CompensateLensDistortionExp2

	{attribute 'TcIecLibraryType'}
	{attribute 'external_name' := 'F_VN_CompensateLensDistortionExp2_GUID_D58090D3_3F13_0BD1_6EF1_2A37C7563873'}
	(* Transforms an image to compensate the lens distortion. (expert function) *)
	FUNCTION F_VN_CompensateLensDistortionExp2 : HRESULT
	VAR_INPUT
		ipSrcImage	:	ITcVnImage;	(* Source image *)
		ipDestImage	:	REFERENCE TO ITcVnImage;	(* Destination image (An appropriate destination image will be created if required.) *)
		aCameraMatrix	:	REFERENCE TO TcVnMatrix3x3_LREAL;	(* Camera matrix containing the intrinsic parameters *)
		aDistortionCoefficients	:	REFERENCE TO TcVnArray8_LREAL;	(* Lens distortion coefficients [k1, k2, p1, p2, k3, k4, k5, k6] *)
		aNewCameraMatrix	:	REFERENCE TO TcVnMatrix3x3_LREAL;	(* Allows additional scaling and shifting of the result image *)
		hrPrev	:	HRESULT;	(* HRESULT indicating the result of previous operations (If SUCCEEDED(hrPrev) equals false, no operation is executed.) *)
	END_VAR

END_FUNCTION

// Functions/Geometric and Coordinate Transformations/Calibration/F_VN_CompensateLensDistortionForPoints

	{attribute 'TcIecLibraryType'}
	{attribute 'external_name' := 'F_VN_CompensateLensDistortionForPoints_GUID_0DFE1234_C1BF_0BE5_76D0_05221A2F0719'}
	(* Transforms point coordinates to compensate the lens distortion. *)
	FUNCTION F_VN_CompensateLensDistortionForPoints : HRESULT
	VAR_INPUT
		ipSrcPoints	:	ITcVnContainer;	(* Container with source point coordinates (ContainerType_Vector_TcVnPoint2_REAL or ContainerType_Vector_TcVnPoint2_DINT) *)
		ipDestPoints	:	REFERENCE TO ITcVnContainer;	(* Returns a container with the transformed point coordinates (ContainerType_Vector_TcVnPoint2_REAL) *)
		aCameraMatrix	:	REFERENCE TO TcVnMatrix3x3_LREAL;	(* Camera matrix containing the intrinsic parameters *)
		aDistortionCoefficients	:	REFERENCE TO TcVnArray4_LREAL;	(* Lens distortion coefficients [k1, k2, p1, p2] *)
		hrPrev	:	HRESULT;	(* HRESULT indicating the result of previous operations (If SUCCEEDED(hrPrev) equals false, no operation is executed.) *)
	END_VAR

END_FUNCTION

// Functions/Geometric and Coordinate Transformations/Calibration/F_VN_CompensateLensDistortionForPointsExp1

	{attribute 'TcIecLibraryType'}
	{attribute 'external_name' := 'F_VN_CompensateLensDistortionForPointsExp1_GUID_6C0BC580_C288_0BCD_47F2_2ABBC33EAC97'}
	(* Transforms point coordinates to compensate the lens distortion. (expert function) *)
	FUNCTION F_VN_CompensateLensDistortionForPointsExp1 : HRESULT
	VAR_INPUT
		ipSrcPoints	:	ITcVnContainer;	(* Container with source point coordinates (ContainerType_Vector_TcVnPoint2_REAL or ContainerType_Vector_TcVnPoint2_DINT) *)
		ipDestPoints	:	REFERENCE TO ITcVnContainer;	(* Returns a container with the transformed point coordinates (ContainerType_Vector_TcVnPoint2_REAL) *)
		aCameraMatrix	:	REFERENCE TO TcVnMatrix3x3_LREAL;	(* Camera matrix containing the intrinsic parameters *)
		aDistortionCoefficients	:	REFERENCE TO TcVnArray8_LREAL;	(* Lens distortion coefficients [k1, k2, p1, p2, k3, k4, k5, k6] *)
		hrPrev	:	HRESULT;	(* HRESULT indicating the result of previous operations (If SUCCEEDED(hrPrev) equals false, no operation is executed.) *)
	END_VAR

END_FUNCTION

// Functions/Geometric and Coordinate Transformations/Calibration/F_VN_CompensateLensDistortionForPointsExp2

	{attribute 'TcIecLibraryType'}
	{attribute 'external_name' := 'F_VN_CompensateLensDistortionForPointsExp2_GUID_23DA916F_77FF_01F9_6576_A41D23115D42'}
	(* Transforms point coordinates to compensate the lens distortion. (expert function) *)
	FUNCTION F_VN_CompensateLensDistortionForPointsExp2 : HRESULT
	VAR_INPUT
		ipSrcPoints	:	ITcVnContainer;	(* Container with source point coordinates (ContainerType_Vector_TcVnPoint2_REAL or ContainerType_Vector_TcVnPoint2_DINT) *)
		ipDestPoints	:	REFERENCE TO ITcVnContainer;	(* Returns a container with the transformed point coordinates (ContainerType_Vector_TcVnPoint2_REAL) *)
		aCameraMatrix	:	REFERENCE TO TcVnMatrix3x3_LREAL;	(* Camera matrix containing the intrinsic parameters *)
		aDistortionCoefficients	:	REFERENCE TO TcVnArray8_LREAL;	(* Lens distortion coefficients [k1, k2, p1, p2, k3, k4, k5, k6] *)
		aNewCameraMatrix	:	REFERENCE TO TcVnMatrix3x3_LREAL;	(* Allows additional shifting of the result point coordinates *)
		hrPrev	:	HRESULT;	(* HRESULT indicating the result of previous operations (If SUCCEEDED(hrPrev) equals false, no operation is executed.) *)
	END_VAR

END_FUNCTION

// Functions/Geometric and Coordinate Transformations/Calibration/F_VN_DetectPatternPoints

	{attribute 'TcIecLibraryType'}
	{attribute 'external_name' := 'F_VN_DetectPatternPoints_GUID_F635E589_132F_0D5F_6901_B9B13A70F175'}
	(* Detects calibration pattern points (circles) within the provided image. *)
	FUNCTION F_VN_DetectPatternPoints : HRESULT
	VAR_INPUT
		ipSrcImage	:	ITcVnImage;	(* Source image (USINT, 1 channel) *)
		ipPatternPoints	:	REFERENCE TO ITcVnContainer;	(* Returns the pattern point positions (ContainerType_Vector_TcVnPoint2_REAL; Non-zero interface pointers are reused.) *)
		stBlobDetectionParams	:	REFERENCE TO TcVnParamsBlobDetection;	(* Parameters to detect and filter contours. *)
		nNumberOfPoints	:	UDINT;	(* Expected number of pattern points *)
		hrPrev	:	HRESULT;	(* HRESULT indicating the result of previous operations (If SUCCEEDED(hrPrev) equals false, no operation is executed.) *)
	END_VAR

END_FUNCTION

// Functions/Geometric and Coordinate Transformations/Calibration/F_VN_DetectPatternPointsExp

	{attribute 'TcIecLibraryType'}
	{attribute 'external_name' := 'F_VN_DetectPatternPointsExp_GUID_185A9E39_7461_030E_7EC8_A1CD6A0AD49D'}
	(* Detects calibration pattern points (circles) within the provided image. (expert function) *)
	FUNCTION F_VN_DetectPatternPointsExp : HRESULT
	VAR_INPUT
		ipSrcImage	:	ITcVnImage;	(* Source image (USINT, 1 channel) *)
		ipPatternPoints	:	REFERENCE TO ITcVnContainer;	(* Returns the pattern point positions (ContainerType_Vector_TcVnPoint2_REAL; Non-zero interface pointers are reused.) *)
		stBlobDetectionParams	:	REFERENCE TO TcVnParamsBlobDetection;	(* Parameters to detect and filter contours. *)
		nNumberOfPoints	:	UDINT;	(* Expected number of pattern points *)
		fSizeDiffThresFactor	:	REAL;	(* Threshold for filtering contours by average size *)
		bSubpixelAccuracy	:	BOOL;	(* If true, the pattern points are detected with subpixel accuracy *)
		eEdgeDirection	:	ETcVnEdgeDirection;	(* Specification of the edge direction to search for (from center to outside circle) *)
		fMinStrength	:	REAL;	(* Specification of the minimum strength (intensity difference) of the edge to search for *)
		nMaxThickness	:	UDINT;	(* Specification of the maximum thickness of the edge to search for, which means fMinStrength must be reached within nMaxThickness pixels *)
		nSubpixelsIterations	:	UDINT;	(* Specifies the number of subpixels (for INTERPOLATION, 10 - 20 usually is sufficient) or maximum number of iterations for optimizing the parameters (for APPROX_ERF and APPROX_GAUSSIAN, 50 - 100 usually is sufficient) *)
		nSearchLines	:	UDINT;	(* Specifies the amount of search lines, which are equally distributed in all directions (must be >= 8 and a multiple of 4) *)
		fApproxPrecision	:	REAL;	(* Specifies the approximation precision for APPROX_ERF and APPROX_GAUSSIAN (0.001 usually is sufficient, unused for INTERPOLATION) *)
		eAlgorithm	:	ETcVnEdgeDetectionAlgorithm;	(* Selection of the edge detection algorithm *)
		hrPrev	:	HRESULT;	(* HRESULT indicating the result of previous operations (If SUCCEEDED(hrPrev) equals false, no operation is executed.) *)
	END_VAR

END_FUNCTION

// Functions/Geometric and Coordinate Transformations/Calibration/F_VN_GenerateCalibrationPatternReferencePoints

	{attribute 'TcIecLibraryType'}
	{attribute 'external_name' := 'F_VN_GenerateCalibrationPatternReferencePoints_GUID_4E159D61_A898_06C9_628A_D45D7C91F334'}
	(* Generate reference points for common calibration patterns. *)
	FUNCTION F_VN_GenerateCalibrationPatternReferencePoints : HRESULT
	VAR_INPUT
		ipReferencePoints	:	REFERENCE TO ITcVnContainer;	(* Returns the generated reference points (ContainerType_Vector_TcVnPoint3_REAL) *)
		ePattern	:	ETcVnCalibrationPattern;	(* Calibration pattern type *)
		eOrigin	:	ETcVnCalibrationPatternOrigin;	(* Calibration pattern origin *)
		nWidth	:	UDINT;	(* Pattern width, i.e. number of pattern points in x direction *)
		nHeight	:	UDINT;	(* Pattern height, i.e. number of pattern points in y direction *)
		fDistX	:	REAL;	(* Distance between pattern points in x direction *)
		fDistY	:	REAL;	(* Distance between pattern points in y direction *)
		hrPrev	:	HRESULT;	(* HRESULT indicating the result of previous operations (If SUCCEEDED(hrPrev) equals false, no operation is executed.) *)
	END_VAR

END_FUNCTION

// Functions/Geometric and Coordinate Transformations/Calibration/F_VN_ImagePointsWorldDistance

	{attribute 'TcIecLibraryType'}
	{attribute 'external_name' := 'F_VN_ImagePointsWorldDistance_GUID_10D72248_8801_0A3B_5697_703873EDFC6F'}
	(* Computes the distance in the world coordinate system between two points (in the same world coordinate z layer) given in image coordinates. *)
	FUNCTION F_VN_ImagePointsWorldDistance : HRESULT
	VAR_INPUT
		aImagePoint1	:	REFERENCE TO TcVnPoint2_REAL;	(* First point in the image coordinate system *)
		aImagePoint2	:	REFERENCE TO TcVnPoint2_REAL;	(* Second point in the image coordinate system *)
		fWorldDistance	:	REFERENCE TO LREAL;	(* Returns the distance between aImagePoint1 and aImagePoint2 in the world coordinate system *)
		aCameraMatrix	:	REFERENCE TO TcVnMatrix3x3_LREAL;	(* 3x3 camera matrix containing the intrinsic parameters *)
		aDistortionCoefficients	:	REFERENCE TO TcVnArray8_LREAL;	(* Lens distortion coefficients [k1, k2, p1, p2, k3, k4, k5, k6] *)
		aRotationMatrix	:	REFERENCE TO TcVnMatrix3x3_LREAL;	(* 3x3 rotation matrix *)
		aTranslationVector	:	REFERENCE TO TcVnVector3_LREAL;	(* Translation vector *)
		fZ	:	LREAL;	(* z coordinate (world coordinate system) of the given points (0 would be at (toplevel) calibration pattern) *)
		hrPrev	:	HRESULT;	(* HRESULT indicating the result of previous operations (If SUCCEEDED(hrPrev) equals false, no operation is executed.) *)
	END_VAR

END_FUNCTION

// Functions/Geometric and Coordinate Transformations/Calibration/F_VN_SortDetectedPatternPoints

	{attribute 'TcIecLibraryType'}
	{attribute 'external_name' := 'F_VN_SortDetectedPatternPoints_GUID_B29C960B_DD9F_05B7_7B79_9632692FB44E'}
	(* Sort the detected pattern points according to the relative positions of the calibration pattern points. *)
	FUNCTION F_VN_SortDetectedPatternPoints : HRESULT
	VAR_INPUT
		ipImagePoints	:	ITcVnContainer;	(* Detected pattern point positions in the image coordinate system (will be sorted by this function, ContainerType_Vector_TcVnPoint2_REAL) *)
		ipPatternPoints	:	ITcVnContainer;	(* The pattern points in the calibration pattern coordinate system, used as a reference to sort ipImagePoints (ContainerType_Vector_TcVnPoint3_REAL) *)
		hrPrev	:	HRESULT;	(* HRESULT indicating the result of previous operations (If SUCCEEDED(hrPrev) equals false, no operation is executed.) *)
	END_VAR

END_FUNCTION

// Functions/Geometric and Coordinate Transformations/Calibration/F_VN_TransformCoordinatesPlanar_Container

	{attribute 'TcIecLibraryType'}
	{attribute 'external_name' := 'F_VN_TransformCoordinatesPlanar_Container_GUID_70DB80CA_A0FF_00B4_56DB_469AF1A061D6'}
	(* Compute real-world coordinates for given image points or vice versa. *)
	FUNCTION F_VN_TransformCoordinatesPlanar_Container : HRESULT
	VAR_INPUT
		ipSrcPoints	:	ITcVnContainer;	(* Container with 2D source points (TcVnPoint2_DINT or TcVnPoint2_REAL or TcVnPoint2_LREAL) *)
		ipDestPoints	:	REFERENCE TO ITcVnContainer;	(* Returns the transformed 2D points (TcVnPoint2_LREAL) *)
		aTransformationMatrix	:	REFERENCE TO TcVnMatrix3x3_LREAL;	(* Transformation matrix obtained with VnCalibrateCameraPlanar() or its inverse matrix obtained with VnInvertMatrix3x3() *)
		hrPrev	:	HRESULT;	(* HRESULT indicating the result of previous operations (If SUCCEEDED(hrPrev) equals false, no operation is executed.) *)
	END_VAR

END_FUNCTION

// Functions/Geometric and Coordinate Transformations/Calibration/F_VN_TransformCoordinatesPlanar_Point

	{attribute 'TcIecLibraryType'}
	{attribute 'external_name' := 'F_VN_TransformCoordinatesPlanar_Point_GUID_84213DD6_8F0C_035E_5807_9708C5FFE02C'}
	(* Compute real-world coordinates for a given image point or vice versa. *)
	FUNCTION F_VN_TransformCoordinatesPlanar_Point : HRESULT
	VAR_INPUT
		aSrcPoint	:	REFERENCE TO TcVnPoint2_LREAL;	(* Point in the source coordinate system *)
		aDestPoint	:	REFERENCE TO TcVnPoint2_LREAL;	(* Returns point in the destination coordinate system *)
		aTransformationMatrix	:	REFERENCE TO TcVnMatrix3x3_LREAL;	(* Transformation matrix obtained with VnCalibrateCameraPlanar() or its inverse matrix obtained with VnInvertMatrix3x3() *)
		hrPrev	:	HRESULT;	(* HRESULT indicating the result of previous operations (If SUCCEEDED(hrPrev) equals false, no operation is executed.) *)
	END_VAR

END_FUNCTION

// Functions/Geometric and Coordinate Transformations/Calibration/F_VN_TransformCoordinatesImageToWorld_Container

	{attribute 'TcIecLibraryType'}
	{attribute 'external_name' := 'F_VN_TransformCoordinatesImageToWorld_Container_GUID_434C253F_D489_0111_69F1_8ECF0859939C'}
	(* Transform 2D image point coordinates to 3D world coordinates (using intrinsic + extrinsic calibration results). *)
	FUNCTION F_VN_TransformCoordinatesImageToWorld_Container : HRESULT
	VAR_INPUT
		ipSrcPoints2D	:	ITcVnContainer;	(* Container with 2D source points (TcVnPoint2_DINT or TcVnPoint2_REAL or TcVnPoint2_LREAL) *)
		ipDestPoints3D	:	REFERENCE TO ITcVnContainer;	(* Returns the transformed 3D points (TcVnPoint3_LREAL) *)
		aCameraMatrix	:	REFERENCE TO TcVnMatrix3x3_LREAL;	(* 3x3 camera matrix containing the intrinsic parameters *)
		aDistortionCoefficients	:	REFERENCE TO TcVnArray8_LREAL;	(* Lens distortion coefficients [k1, k2, p1, p2, k3, k4, k5, k6] *)
		aRotationMatrix	:	REFERENCE TO TcVnMatrix3x3_LREAL;	(* 3x3 rotation matrix *)
		aTranslationVector	:	REFERENCE TO TcVnVector3_LREAL;	(* Translation vector *)
		fZ	:	LREAL;	(* z coordinate (world coordinate system) of the transformed points (0 would be at (toplevel) calibration pattern) *)
		hrPrev	:	HRESULT;	(* HRESULT indicating the result of previous operations (If SUCCEEDED(hrPrev) equals false, no operation is executed.) *)
	END_VAR

END_FUNCTION

// Functions/Geometric and Coordinate Transformations/Calibration/F_VN_TransformCoordinatesImageToWorld_Point

